// TwinCAT 3 PLC project EngineeringToolbox
// Title: EngineeringToolbox
// Company: Beckhoff Electronics Mfg
// Author: Daniel Schlingmann
// ProjectVersion: 3.1.2.4
// Description: Engineering Toolbox Library The library is provided "as-is" for TwinCAT3.1 by the Beckhoff Industry Management for Electronics Manufacturing. Please check the function "DisclaimerStatement : WSTRING[1500]" in additon to the following disclaimer: THE SOFTWARE IS PROVIDED "AS IS", WITHOUT WARRANTY OF ANY KIND, EXPRESS OR IMPLIED, INCLUDING BUT NOT LIMITED TO THE WARRANTIES OF MERCHANTABILITY, FITNESS FOR A PARTICULAR PURPOSE AND NONINFRINGEMENT. IN NO EVENT SHALL THE AUTHORS OR COPYRIGHT HOLDERS BE LIABLE FOR ANY CLAIM, DAMAGES OR OTHER LIABILITY, WHETHER IN AN ACTION OF CONTRACT, TORT OR OTHERWISE, ARISING FROM, OUT OF OR IN CONNECTION WITH THE SOFTWARE OR THE USE OR OTHER DEALINGS IN THE SOFTWARE.
// ProgramVersion: 3.1.4022.7
// libraries:
//   Tc2_Drive, * (Beckhoff Automation GmbH)
//   Tc2_EtherCAT, * (Beckhoff Automation GmbH)
//   Tc2_IoFunctions, * (Beckhoff Automation GmbH)
//   Tc2_Math, * (Beckhoff Automation GmbH)
//   Tc2_MC2, * (Beckhoff Automation GmbH)
//   Tc2_MC2_Camming, * (Beckhoff Automation GmbH)
//   Tc2_MC2_Drive, * (Beckhoff Automation GmbH)
//   Tc2_MC2_FlyingSaw, * (Beckhoff Automation GmbH)
//   Tc2_MDP, * (Beckhoff Automation GmbH)
//   Tc2_ModbusRTU, * (Beckhoff Automation GmbH)
//   Tc2_ModbusSrv, * (Beckhoff Automation GmbH)
//   Tc2_NC, * (Beckhoff Automation GmbH)
//   Tc2_NCI, * (Beckhoff Automation GmbH)
//   Tc2_NcKinematicTransformation, * (Beckhoff Automation GmbH)
//   Tc2_PlcInterpolation, * (Beckhoff Automation GmbH)
//   Tc2_SerialCom, * (Beckhoff Automation GmbH)
//   Tc2_Smtp, * (Beckhoff Automation GmbH)
//   Tc2_Standard, * (Beckhoff Automation GmbH)
//   Tc2_SUPS, * (Beckhoff Automation GmbH)
//   Tc2_System, * (Beckhoff Automation GmbH)
//   Tc2_TcpIp, * (Beckhoff Automation GmbH)
//   Tc2_Utilities, * (Beckhoff Automation GmbH)
//   Tc2_XmlDataSrv, * (Beckhoff Automation GmbH)
//   Tc3_Module, * (Beckhoff Automation GmbH)
//   Tc2_BackupRestoreEL6900,newest,Beckhoff Automation GmbH
// project tree:
//   GVLs/ Gvl.TcGVL (not stored), PARAM.TcGVL (not stored)
//   POUs/BoundsCheck/ boundsError.TcPOU (not stored), boundsOK.TcPOU (not stored), checkBounds.TcPOU (not stored), CheckBoundsInfo.TcPOU (not stored)
//   POUs/Connectivity/ADS/ AdsDataExchange.TcPOU (not stored)
//   POUs/Connectivity/ Ipv4Addr_TO_UDINT.TcPOU (not stored), U_DEVICE_COM_CACHE.TcDUT (not stored), U_IPv4Addr.TcDUT, isValidIPv4Addr.TcPOU (not stored)
//   POUs/Connectivity/TF6310-TcpServer/DeviceCom/ TCPDeviceCom_SendRecBytes.TcPOU (not stored), TCPDeviceCom_SendRecString.TcPOU (not stored)
//   POUs/Connectivity/TF6340-SerialCom/ComPortDeviceCom/ ComPortDeviceCom_BufferHandle.TcPOU (not stored), ComPortDeviceCom_SendRecBytes.TcPOU (not stored), ComPortDeviceCom_SendRecString.TcPOU, ComPortEL6x22BEasyConnect.TcPOU
//   POUs/Connectivity/TF6340-SerialCom/ComPortBasic/ ComPortBackground.TcPOU, ComPortSendRec.TcPOU (not stored)
//   POUs/Connectivity/TF625x-Modbus/Master/TF6250-ModbusTcpServer/TCP/ ModbusTcpMaster.TcPOU
//   POUs/Connectivity/TF625x-Modbus/Master/TF6250-ModbusTcpServer/UDP/ ModbusUdpMaster.TcPOU (not stored)
//   POUs/Connectivity/TF625x-Modbus/Master/TF6255-ModbusRtu/ ModbusRtuMaster22B.TcPOU, ModbusRtuMaster5B.TcPOU, ModbusRtuMasterPC.TcPOU (not stored)
//   POUs/Connectivity/TF625x-Modbus/Master/_Components/ ModbusJob.TcPOU (not stored), ModbusSlaveCom.TcPOU (not stored)
//   POUs/Connectivity/TF625x-Modbus/Slave/ ModbusSlaveBase.TcPOU (not stored)
//   POUs/Connectivity/TF6310-TcpServer/TcpBasic/ TCPSendRecCtrl.TcPOU, TCPConnectionCtrl.TcPOU (not stored), TCPSocketCtrl.TcPOU (not stored)
//   POUs/Connectivity/TF6310-TcpServer/UdpBasic/ UDPSendRecCtrl.TcPOU (not stored), UDPServerCtrl.TcPOU, UDPSocketCtrl.TcPOU (not stored)
//   POUs/ControllerTools/ AverageFilter.TcPOU (not stored), PIDController.TcPOU, PT1Filter.TcPOU (not stored), signum.TcPOU, SlewRateLimitter.TcPOU (not stored), SlidingAverageExt.TcPOU (not stored), SlidingAverage.TcPOU (not stored), ThreePointController.TcPOU (not stored)
//   POUs/DataBuffer/ DoubleBuffer.TcPOU, Quicksort.TcPOU
//   POUs/DataBuffer/FiFo/ Fifo.TcPOU, FiFoExt.TcPOU, FiFoLRealSimple.TcPOU, FiFoBase.TcPOU (not stored)
//   POUs/DataBuffer/LiFo/ LiFoBase.TcPOU (not stored), LiFoExt.TcPOU, LiFo.TcPOU (not stored)
//   POUs/DataBuffer/Ringbuffer/ RingbufferBase.TcPOU (not stored), Ringbuffer.TcPOU, RingbufferCharSimple.TcPOU, RingbufferExt.TcPOU (not stored), RingbufferByteSimple.TcPOU, RingbufferLRealSimple.TcPOU (not stored), RingbufferRealSimple.TcPOU (not stored)
//   POUs/EventLogger/ EventsWriteToLogbook.TcPOU (not stored), EVENT_HANDLING_CONFIG.TcDUT, getEventClassPriority.TcPOU (not stored), getEventClassText.TcPOU (not stored), SOURCE_ID.TcDUT
//   POUs/EventLogger/ReadEvents/ EventlogRead.TcPOU (not stored), EVENTLOG_READ_DATA.TcDUT, EVENTLOG_READ_HANDLEINFO.TcDUT, EVENTLOG_READ_STREAM.TcDUT (not stored), EVENTLOG_READ_STREAM_DATA_RAW.TcDUT (not stored), EVENTLOG_READ_STREAM_DATA_RAW_EX.TcDUT (not stored)
//   POUs/EventLogger/TriggerEvents/ EventHandling.TcPOU (not stored), EventHandlingGrp10.TcPOU (not stored), EventHandlingGrp25.TcPOU (not stored), EventHandlingGrp50.TcPOU, EventHandlingGrpCustomized.TcPOU (not stored), EventHandlingConfirmIsReq.TcPOU (not stored), EventHandlingStatisticInfo.TcPOU (not stored)
//   POUs/Fieldbus/CANopen/ CANopenMasterDiag.TcPOU, CANopenMasterIO.TcPOU (not stored)
//   POUs/Fieldbus/EAP/ EAP_PUB_SUB_IO.TcPOU (not stored), EAP_DEVICE_IO.TcPOU, EAP_PUB_VAR.TcPOU (not stored), EAP_SUB_VAR.TcPOU
//   POUs/Fieldbus/EtherCAT/ EcCoEReadNewestDiagMsg.TcPOU (not stored), EcDiagBase.TcPOU (not stored), EcDiagBase_wEvents.TcPOU (not stored)
//   POUs/Fieldbus/EtherCAT/_Components/ EcMasterIO.TcPOU, EcMasterSupervisor.TcPOU (not stored), EcSlavesDiag.TcPOU (not stored), EcSlaveSupervisor.TcPOU (not stored), EC_MASTER_DEVICE_STATE.TcDUT (not stored), EC_SLAVE_DIAG_INFO_DATA.TcDUT (not stored)
//   POUs/Fieldbus/Profibus/ ProfibusMasterDiag.TcPOU (not stored), ProfibusMasterIO.TcPOU (not stored)
//   POUs/Fieldbus/Profinet/ ProfinetControllerIO.TcPOU (not stored), ProfinetControllerIO_wEvents.TcPOU (not stored), ProfinetDeviceIO.TcPOU (not stored)
//   POUs/FileHandling/Basic/ FileHandling.TcPOU (not stored), ReadDirSimple.TcPOU (not stored), ReadDirSimpleExt.TcPOU (not stored)
//   POUs/FileHandling/TF6421-XmlServer/ XmlReadWrite.TcPOU (not stored), XmlReadWriteWithBackupFile.TcPOU
//   POUs/IO/Analog/ AnalogIn.TcPOU (not stored), AnalogIn32.TcPOU (not stored), AnalogInELMBase.TcPOU, AnalogInELMSingleSampleDINT.TcPOU (not stored), AnalogInELMSingleSampleREAL.TcPOU (not stored), AnalogInREAL.TcPOU (not stored), AnalogOut.TcPOU (not stored)
//   POUs/IO/ BlowOffSensors.TcPOU (not stored), Button.TcPOU (not stored), ButtonExt.TcPOU (not stored), Fuse.TcPOU, InOut.TcPOU, InOutExt.TcPOU (not stored), Input.TcPOU, Output.TcPOU (not stored)
//   POUs/IO/Cylinder/ Cylinder.TcPOU, CylinderExt.TcPOU (not stored), CylinderType4.TcPOU, I_Cylinder.TcIO
//   POUs/IO/Drives/ AxDriveBase.TcPOU (not stored), AxDriveGetRef.TcPOU (not stored), I_AxDriveBase.TcIO (not stored)
//   POUs/IO/Drives/CoE/ AxDriveCoE.TcPOU, AxDriveCoE_wEvents.TcPOU (not stored), CiA_DS402Controlword.TcPOU (not stored), CiA_DS402Statusword.TcPOU, eCiA_DS402_CONTROL_CMD.TcDUT (not stored), eCiA_DS402_STATUS_STATE.TcDUT (not stored)
//   POUs/IO/Drives/CoE/EL72xx/ AxDriveCoE_EL72xxParam.TcPOU, CiA_DS402StatuswordEx7xxx.TcPOU (not stored)
//   POUs/IO/Drives/DC/Ey73xx/ AxDriveDC.TcPOU (not stored), AxDriveDC_wEvents.TcPOU (not stored)
//   POUs/IO/Drives/SoE/ AxDriveSoE_Ax5000CommutationCalib.TcPOU, AxDriveSoE_Ax5000CalcPower.TcPOU (not stored), AxDriveSoE_Ax5000SwitchParamSet.TcPOU, Ax580x.TcPOU (not stored), AxDriveSoE_Ax5000.TcPOU (not stored), AxDriveSoE_Ax5000Param.TcPOU (not stored), AxDriveSoE_Ax5000wEvents.TcPOU (not stored), AxDriveSoE_Rexroth.TcPOU (not stored)
//   POUs/IO/Drives/SoE/Ax5000ParamSTRUCTs/P/ AX5000_P_0001.TcDUT, AX5000_P_0002.TcDUT, AX5000_P_0003.TcDUT, AX5000_P_0004.TcDUT, AX5000_P_0009.TcDUT (not stored), AX5000_P_0010.TcDUT (not stored), AX5000_P_0020.TcDUT (not stored), AX5000_P_0021.TcDUT (not stored), AX5000_P_0040.TcDUT (not stored), AX5000_P_0050.TcDUT (not stored), AX5000_P_0051.TcDUT (not stored), AX5000_P_0052.TcDUT (not stored), AX5000_P_0053.TcDUT (not stored), AX5000_P_0054.TcDUT, AX5000_P_0055.TcDUT, AX5000_P_0056.TcDUT (not stored), AX5000_P_0057.TcDUT (not stored), AX5000_P_0058.TcDUT (not stored), AX5000_P_0059.TcDUT (not stored), AX5000_P_0060.TcDUT, AX5000_P_0061.TcDUT (not stored), AX5000_P_0062.TcDUT, AX5000_P_0063.TcDUT (not stored), AX5000_P_0064.TcDUT, AX5000_P_0065.TcDUT (not stored), AX5000_P_0066.TcDUT (not stored), AX5000_P_0067.TcDUT (not stored), AX5000_P_0068.TcDUT, AX5000_P_0069.TcDUT (not stored), AX5000_P_0070.TcDUT (not stored), AX5000_P_0071.TcDUT (not stored), AX5000_P_0072.TcDUT (not stored), AX5000_P_0073.TcDUT (not stored), AX5000_P_0074.TcDUT, AX5000_P_0075.TcDUT, AX5000_P_0076.TcDUT, AX5000_P_0077.TcDUT, AX5000_P_0078.TcDUT (not stored), AX5000_P_0088.TcDUT (not stored), AX5000_P_0089.TcDUT, AX5000_P_0090.TcDUT, AX5000_P_0091.TcDUT, AX5000_P_0092.TcDUT (not stored), AX5000_P_0093.TcDUT (not stored), AX5000_P_0096.TcDUT, AX5000_P_0097.TcDUT (not stored), AX5000_P_0098_beckhoff.TcDUT, AX5000_P_0098_beckhoff_electrical_data.TcDUT, AX5000_P_0099.TcDUT, AX5000_P_0100.TcDUT, AX5000_P_0101.TcDUT (not stored), AX5000_P_0102.TcDUT (not stored), AX5000_P_0103.TcDUT, AX5000_P_0104.TcDUT (not stored), AX5000_P_0105.TcDUT, AX5000_P_0106.TcDUT (not stored), AX5000_P_0107.TcDUT, AX5000_P_0108.TcDUT (not stored), AX5000_P_0109.TcDUT, AX5000_P_0110.TcDUT (not stored), AX5000_P_0111.TcDUT, AX5000_P_0112.TcDUT, AX5000_P_0113.TcDUT (not stored), AX5000_P_0114.TcDUT (not stored), AX5000_P_0115.TcDUT, AX5000_P_0116.TcDUT (not stored), AX5000_P_0117.TcDUT, AX5000_P_0118.TcDUT (not stored), AX5000_P_0119.TcDUT (not stored), AX5000_P_0125.TcDUT (not stored), AX5000_P_0126.TcDUT (not stored), AX5000_P_0127.TcDUT (not stored), AX5000_P_0128.TcDUT (not stored), AX5000_P_0150.TcDUT (not stored), AX5000_P_0151.TcDUT, AX5000_P_0152.TcDUT (not stored), AX5000_P_0153.TcDUT, AX5000_P_0154.TcDUT (not stored), AX5000_P_0155.TcDUT, AX5000_P_0158.TcDUT (not stored), AX5000_P_0159.TcDUT (not stored), AX5000_P_0160.TcDUT (not stored), AX5000_P_0161.TcDUT (not stored), AX5000_P_0162.TcDUT (not stored), AX5000_P_0163.TcDUT (not stored), AX5000_P_0165.TcDUT, AX5000_P_0166.TcDUT (not stored), AX5000_P_0167.TcDUT, AX5000_P_0168.TcDUT, AX5000_P_0169.TcDUT (not stored), AX5000_P_0170.TcDUT (not stored), AX5000_P_0171.TcDUT, AX5000_P_0180.TcDUT (not stored), AX5000_P_0181.TcDUT (not stored), AX5000_P_0182.TcDUT, AX5000_P_0183.TcDUT (not stored), AX5000_P_0184.TcDUT (not stored), AX5000_P_0185.TcDUT, AX5000_P_0188.TcDUT (not stored), AX5000_P_0189.TcDUT (not stored), AX5000_P_0192.TcDUT, AX5000_P_0193.TcDUT, AX5000_P_0196.TcDUT (not stored), AX5000_P_0198.TcDUT (not stored), AX5000_P_0199.TcDUT, AX5000_P_0200.TcDUT (not stored), AX5000_P_0201.TcDUT (not stored), AX5000_P_0202.TcDUT (not stored), AX5000_P_0203.TcDUT (not stored), AX5000_P_0204.TcDUT (not stored), AX5000_P_0205.TcDUT (not stored), AX5000_P_0206.TcDUT (not stored), AX5000_P_0207.TcDUT (not stored), AX5000_P_0208.TcDUT (not stored), AX5000_P_0209.TcDUT (not stored), AX5000_P_0210.TcDUT (not stored), AX5000_P_0211.TcDUT (not stored), AX5000_P_0212.TcDUT (not stored), AX5000_P_0213.TcDUT (not stored), AX5000_P_0214.TcDUT (not stored), AX5000_P_0215.TcDUT (not stored), AX5000_P_0216.TcDUT, AX5000_P_0217.TcDUT (not stored), AX5000_P_0218.TcDUT, AX5000_P_0219.TcDUT (not stored), AX5000_P_0220.TcDUT (not stored), AX5000_P_0221.TcDUT, AX5000_P_0250.TcDUT, AX5000_P_0251.TcDUT (not stored), AX5000_P_0252.TcDUT (not stored), AX5000_P_0253.TcDUT (not stored), AX5000_P_0254.TcDUT (not stored), AX5000_P_0255.TcDUT (not stored), AX5000_P_0256.TcDUT (not stored), AX5000_P_0270.TcDUT (not stored), AX5000_P_0271.TcDUT, AX5000_P_0272.TcDUT, AX5000_P_0273.TcDUT (not stored), AX5000_P_0274.TcDUT (not stored), AX5000_P_0275.TcDUT (not stored), AX5000_P_0276.TcDUT (not stored), AX5000_P_0277.TcDUT, AX5000_P_0278.TcDUT, AX5000_P_0300.TcDUT, AX5000_P_0301.TcDUT (not stored), AX5000_P_0302.TcDUT (not stored), AX5000_P_0303.TcDUT (not stored), AX5000_P_0304.TcDUT (not stored), AX5000_P_0305.TcDUT (not stored), AX5000_P_0306.TcDUT, AX5000_P_0307.TcDUT, AX5000_P_0308.TcDUT (not stored), AX5000_P_0309.TcDUT, AX5000_P_0310.TcDUT (not stored), AX5000_P_0311.TcDUT (not stored), AX5000_P_0312.TcDUT (not stored), AX5000_P_0313.TcDUT (not stored), AX5000_P_0314.TcDUT (not stored), AX5000_P_0315.TcDUT (not stored), AX5000_P_0316.TcDUT (not stored), AX5000_P_0317.TcDUT, AX5000_P_0320.TcDUT (not stored), AX5000_P_0321.TcDUT, AX5000_P_0322.TcDUT, AX5000_P_0323.TcDUT (not stored), AX5000_P_0324.TcDUT (not stored), AX5000_P_0325.TcDUT (not stored), AX5000_P_0326.TcDUT, AX5000_P_0350.TcDUT (not stored), AX5000_P_0351.TcDUT (not stored), AX5000_P_0352.TcDUT (not stored), AX5000_P_0353.TcDUT, AX5000_P_0354.TcDUT (not stored), AX5000_P_0356.TcDUT (not stored), AX5000_P_0360.TcDUT (not stored), AX5000_P_0361.TcDUT, AX5000_P_0400.TcDUT, AX5000_P_0401.TcDUT, AX5000_P_0402.TcDUT (not stored), AX5000_P_0451.TcDUT (not stored), AX5000_P_0452.TcDUT, AX5000_P_0453.TcDUT, AX5000_P_0454.TcDUT (not stored), AX5000_P_0455.TcDUT, AX5000_P_0456.TcDUT (not stored), AX5000_P_0457.TcDUT (not stored), AX5000_P_0458.TcDUT (not stored), AX5000_P_0459.TcDUT (not stored), AX5000_P_0460.TcDUT, AX5000_P_0461.TcDUT (not stored), AX5000_P_0462.TcDUT, AX5000_P_0463.TcDUT, AX5000_P_0464.TcDUT (not stored), AX5000_P_0502.TcDUT, AX5000_P_0503.TcDUT (not stored), AX5000_P_0504.TcDUT (not stored), AX5000_P_0505.TcDUT (not stored), AX5000_P_0511.TcDUT (not stored), AX5000_P_0512.TcDUT (not stored), AX5000_P_0513.TcDUT, AX5000_P_0514.TcDUT (not stored), AX5000_P_0515.TcDUT (not stored), AX5000_P_0516.TcDUT (not stored), AX5000_P_0517.TcDUT (not stored), AX5000_P_0518.TcDUT (not stored), AX5000_P_0552.TcDUT, AX5000_P_0553.TcDUT (not stored), AX5000_P_0554.TcDUT (not stored), AX5000_P_0555.TcDUT, AX5000_P_0556.TcDUT (not stored), AX5000_P_0557.TcDUT (not stored), AX5000_P_0558.TcDUT, AX5000_P_0601.TcDUT (not stored), AX5000_P_0602.TcDUT (not stored), AX5000_P_0610.TcDUT (not stored), AX5000_P_0611.TcDUT, AX5000_P_0800.TcDUT (not stored), AX5000_P_0801.TcDUT (not stored), AX5000_P_0802.TcDUT, AX5000_P_0804.TcDUT (not stored), AX5000_P_0805.TcDUT (not stored), AX5000_P_0806.TcDUT (not stored), AX5000_P_0810.TcDUT, AX5000_P_0811.TcDUT (not stored), AX5000_P_0850.TcDUT (not stored), AX5000_P_0851.TcDUT (not stored), AX5000_P_0900.TcDUT (not stored), AX5000_P_0901.TcDUT, AX5000_P_0902.TcDUT (not stored), AX5000_P_0904.TcDUT, AX5000_P_0905.TcDUT (not stored), AX5000_P_0906.TcDUT, AX5000_P_0912.TcDUT (not stored), AX5000_P_1000.TcDUT (not stored), AX5000_P_1001.TcDUT (not stored), AX5000_P_1002.TcDUT, AX5000_P_1003.TcDUT, AX5000_P_1004.TcDUT (not stored), AX5000_P_1005.TcDUT, AX5000_P_1006.TcDUT, AX5000_P_1007.TcDUT (not stored), AX5000_P_1008.TcDUT (not stored), AX5000_P_1009.TcDUT (not stored), AX5000_P_1010.TcDUT (not stored), AX5000_P_1011.TcDUT, AX5000_P_1012.TcDUT, AX5000_P_1020.TcDUT, AX5000_P_1021.TcDUT, AX5000_P_1022.TcDUT (not stored), AX5000_P_2000.TcDUT (not stored), AX5000_P_2001.TcDUT (not stored), AX5000_P_2002.TcDUT (not stored)
//   POUs/IO/Drives/SoE/Ax5000ParamSTRUCTs/S/ AX5000_S_0001.TcDUT (not stored), AX5000_S_0002.TcDUT, AX5000_S_0007.TcDUT (not stored), AX5000_S_0011.TcDUT (not stored), AX5000_S_0012.TcDUT, AX5000_S_0013.TcDUT (not stored), AX5000_S_0015.TcDUT (not stored), AX5000_S_0016.TcDUT (not stored), AX5000_S_0017.TcDUT, AX5000_S_0018.TcDUT (not stored), AX5000_S_0024.TcDUT (not stored), AX5000_S_0029.TcDUT (not stored), AX5000_S_0030.TcDUT (not stored), AX5000_S_0031.TcDUT (not stored), AX5000_S_0032.TcDUT (not stored), AX5000_S_0033.TcDUT, AX5000_S_0034.TcDUT, AX5000_S_0035.TcDUT (not stored), AX5000_S_0036.TcDUT (not stored), AX5000_S_0037.TcDUT (not stored), AX5000_S_0040.TcDUT, AX5000_S_0043.TcDUT, AX5000_S_0044.TcDUT, AX5000_S_0045.TcDUT, AX5000_S_0046.TcDUT, AX5000_S_0047.TcDUT, AX5000_S_0048.TcDUT (not stored), AX5000_S_0051.TcDUT (not stored), AX5000_S_0053.TcDUT (not stored), AX5000_S_0055.TcDUT (not stored), AX5000_S_0076.TcDUT (not stored), AX5000_S_0079.TcDUT, AX5000_S_0080.TcDUT (not stored), AX5000_S_0081.TcDUT (not stored), AX5000_S_0082.TcDUT (not stored), AX5000_S_0083.TcDUT (not stored), AX5000_S_0084.TcDUT, AX5000_S_0085.TcDUT, AX5000_S_0086.TcDUT (not stored), AX5000_S_0091.TcDUT (not stored), AX5000_S_0092.TcDUT (not stored), AX5000_S_0095.TcDUT (not stored), AX5000_S_0099.TcDUT (not stored), AX5000_S_0100.TcDUT (not stored), AX5000_S_0101.TcDUT (not stored), AX5000_S_0103.TcDUT, AX5000_S_0104.TcDUT (not stored), AX5000_S_0106.TcDUT (not stored), AX5000_S_0107.TcDUT, AX5000_S_0109.TcDUT (not stored), AX5000_S_0110.TcDUT (not stored), AX5000_S_0111.TcDUT (not stored), AX5000_S_0112.TcDUT (not stored), AX5000_S_0113.TcDUT, AX5000_S_0119.TcDUT (not stored), AX5000_S_0120.TcDUT (not stored), AX5000_S_0124.TcDUT (not stored), AX5000_S_0126.TcDUT (not stored), AX5000_S_0130.TcDUT, AX5000_S_0131.TcDUT (not stored), AX5000_S_0134.TcDUT (not stored), AX5000_S_0135.TcDUT (not stored), AX5000_S_0136.TcDUT (not stored), AX5000_S_0137.TcDUT (not stored), AX5000_S_0143.TcDUT (not stored), AX5000_S_0149.TcDUT (not stored), AX5000_S_0159.TcDUT (not stored), AX5000_S_0160.TcDUT (not stored), AX5000_S_0161.TcDUT (not stored), AX5000_S_0162.TcDUT (not stored), AX5000_S_0163.TcDUT (not stored), AX5000_S_0169.TcDUT, AX5000_S_0170.TcDUT, AX5000_S_0179.TcDUT (not stored), AX5000_S_0185.TcDUT (not stored), AX5000_S_0186.TcDUT, AX5000_S_0187.TcDUT (not stored), AX5000_S_0188.TcDUT (not stored), AX5000_S_0189.TcDUT (not stored), AX5000_S_0196.TcDUT, AX5000_S_0200.TcDUT (not stored), AX5000_S_0201.TcDUT (not stored), AX5000_S_0203.TcDUT, AX5000_S_0204.TcDUT, AX5000_S_0206.TcDUT, AX5000_S_0207.TcDUT, AX5000_S_0216.TcDUT (not stored), AX5000_S_0217.TcDUT (not stored), AX5000_S_0219.TcDUT (not stored), AX5000_S_0254.TcDUT (not stored), AX5000_S_0256.TcDUT (not stored), AX5000_S_0257.TcDUT (not stored), AX5000_S_0267.TcDUT (not stored), AX5000_S_0273.TcDUT, AX5000_S_0274.TcDUT (not stored), AX5000_S_0292.TcDUT (not stored), AX5000_S_0295.TcDUT (not stored), AX5000_S_0296.TcDUT (not stored), AX5000_S_0347.TcDUT (not stored), AX5000_S_0348.TcDUT (not stored), AX5000_S_0372.TcDUT (not stored), AX5000_S_0374.TcDUT (not stored), AX5000_S_0375.TcDUT (not stored), AX5000_S_0380.TcDUT (not stored), AX5000_S_0381.TcDUT, AX5000_S_0383.TcDUT (not stored), AX5000_S_0384.TcDUT (not stored), AX5000_S_0390.TcDUT (not stored), AX5000_S_0403.TcDUT, AX5000_S_0405.TcDUT, AX5000_S_0409.TcDUT (not stored), AX5000_S_0410.TcDUT (not stored), AX5000_S_0429.TcDUT (not stored), AX5000_S_0432.TcDUT, AX5000_S_0435.TcDUT (not stored), AX5000_S_0436.TcDUT
//   POUs/IO/Drives/Stepper/ AxDriveStepper.TcPOU (not stored), AxDriveStepperParam.TcPOU (not stored), AxDriveStepper_wEvents.TcPOU (not stored)
//   POUs/IO/EL-EP/ AnalogOut_EL2535.TcPOU (not stored), EL1262_Base.TcPOU, EL3681.TcPOU (not stored), EL1904.TcPOU (not stored), EL69xx.TcPOU (not stored), EL3356.TcPOU, Eyx9xx.TcPOU (not stored), ZB8610.TcPOU (not stored)
//   POUs/IO/EL-EP/EL9x/ EL9501.TcPOU, EL9576.TcPOU (not stored), EL95xxPowerTerminal.TcPOU (not stored), ELSystemTerminal.TcPOU (not stored)
//   POUs/IO/_EcSlaveFWUpdater/ EcSlaveDevFWUpdater.TcPOU (not stored)
//   POUs/IO/_EcSlaveInfoDataIO/ EcSlaveInfoData.TcPOU (not stored), EcSlaveInfoDataExt.TcPOU, I_EcSlaveInfoData.TcIO (not stored)
//   POUs/IO/EL-EP/EL3403/ EL3403.TcPOU (not stored), EL3403Logic.TcPOU (not stored)
//   POUs/IO/EL-EP/EP92xxPwrBox/ EP9214.TcPOU (not stored), EP9214_CHANNEL.TcPOU, EP9224_0037.TcPOU (not stored), EP9224_0037_CHANNEL.TcPOU (not stored)
//   POUs/IO/FreqConv/EtherCAT/DS402/ EcFcDS402_ComBase.TcPOU (not stored)
//   POUs/IO/FreqConv/ IOFcCom.TcPOU (not stored)
//   POUs/IO/Motors/ IOMotor.TcPOU, IOMotor2Dir.TcPOU (not stored), IOMotorStarDelta.TcPOU (not stored)
//   POUs/IO/[underDev]/ Cylinder_wUnitItf.TcPOU (not stored)
//   POUs/IO/_ItfActuators/ I_ActuatorBase.TcIO, I_ActuatorEnableDisable.TcIO, I_ActuatorFwdRev.TcIO (not stored), I_ActuatorFwdBwd.TcIO (not stored), I_ActuatorLeftRight.TcIO (not stored), I_ActuatorOnOff.TcIO (not stored), I_ActuatorOpenClose.TcIO, I_ActuatorPosNeg.TcIO (not stored), I_ActuatorStartStop.TcIO (not stored), I_ActuatorUpDown.TcIO (not stored), I_ActuatorWorkBase.TcIO
//   POUs/IpcDiag/MDP/InfoModuls/ MDP_CPU.TcPOU (not stored), MDP_Fan.TcPOU (not stored), MDP_Mainboard.TcPOU, MDP_RaidSimple.TcPOU (not stored), MDP_ReadModulList.TcPOU, MDP_SiliconDrives.TcPOU (not stored), MDP_UPS.TcPOU
//   POUs/IpcDiag/MDP/ MDP_Info.TcPOU (not stored), MDP_IpcDiag.TcPOU, MDP_IpcDiag_wEvents.TcPOU (not stored)
//   POUs/IpcDiag/ UPSStatus.TcPOU
//   POUs/Logging/ DataFileLogger.TcPOU (not stored), DataUdpLogger.TcPOU, I_LogbookSubscriber.TcIO (not stored), I_Logbook.TcIO (not stored), Logbook.TcPOU (not stored), LogbookData.TcDUT (not stored), LogbookPuplisher.TcPOU (not stored), LogbookSubEventLog.TcPOU (not stored), LogbookSubSendMail.TcPOU (not stored), adsLogError.TcPOU (not stored), adsLogHint.TcPOU, adsLogWarn.TcPOU (not stored), LogbookSubSysLog.TcPOU (not stored), LogbookSubWriteFile.TcPOU (not stored), Logbook_wEventClass.TcPOU (not stored), adsLogwTcEventClass.TcPOU (not stored)
//   POUs/Motion/TF50xx-NC/00_Base/ I_AxNcPTP.TcIO, AxFbBase.TcPOU (not stored), AxRWParaBase.TcPOU (not stored), I_AxNcBase.TcIO (not stored)
//   POUs/Motion/TF50xx-NC/02_Options/Parameter/ AxPara.TcPOU, AxParaCtrl.TcPOU (not stored)
//   POUs/Motion/TF50xx-NC/03_Utilities/ AxAutoWriteSoftLimit.TcPOU (not stored), CoordinateTransformation2D.TcPOU (not stored), AxCalcPosBias.TcPOU (not stored), AxResonanceAvoidance.TcPOU (not stored) (excluded from build), AxSoftSyncDistance.TcPOU (not stored), AxStatemodel.TcPOU (not stored), AxAutoFct.TcPOU, AX_JOB.TcPOU (not stored), getOvrVelo.TcPOU
//   POUs/Motion/TF50xx-NC/ AxNcPTPwJobs.TcPOU (not stored), AxNcBaseExt.TcPOU (not stored), AxNcPtpGear.TcPOU (not stored), AxNcBase.TcPOU (not stored), AxNcPTP.TcPOU
//   POUs/Motion/TF5100-NCI/ NciChannel_wEvents.TcPOU, NciChannel.TcPOU
//   POUs/Motion/TF511x-KIN/03_DUTs/Positions/ KIN_POSITIONS.TcPOU, KIN_POSITIONS_ACS_DUT.TcDUT (not stored), KIN_POSITIONS_MCS_DUT.TcDUT (not stored), U_KIN_POSITIONS.TcDUT (not stored)
//   POUs/Motion/TF511x-KIN/03_DUTs/Trafo/ KIN_CALCTRAFO_AXPOS_PARAM.TcPOU, KIN_STATE_OBSERVER_OID_PARAM.TcPOU, KIN_STATICTRAFO_PARAM.TcPOU (not stored), KIN_TOOLTRAFO_PARAM.TcPOU (not stored), UCS.TcPOU (not stored)
//   POUs/Motion/ VALUE_3D.TcPOU (not stored), VALUE_3D_DUT.TcDUT (not stored), VALUE_6D.TcPOU (not stored), VALUE_6D_DUT.TcDUT (not stored)
//   POUs/Safety/Diag/ SafetyLogicAndIOTerminalDiag.TcPOU (not stored), SafetyIODeviceDiagRead.TcPOU, SafetyIODeviceDiag_wEvents.TcPOU (not stored), SafetyIOsDiag.TcPOU (not stored), SafetyLogicTerminalDiag.TcPOU (not stored), SafetyPlcTerminalDiag.TcPOU (not stored)
//   POUs/StringHelper/ CHR_TO_STR.TcPOU (not stored), cutStrNumberToSeperator.TcPOU, cutStrToSeperator2.TcPOU (not stored), replaceUmlauts.TcPOU (not stored), stringCmp.TcPOU (not stored), STR_TO_ASC.TcPOU, cutStrToSeperator.TcPOU (not stored), cutWStrToSeperator.TcPOU (not stored), DWORD_TO_BINSTR_EXT.TcPOU, DWORD_TO_HEXSTR_EXT.TcPOU (not stored), getCntCharInStr.TcPOU (not stored), getCntCharInWStr.TcPOU (not stored), isWStringNumeric.TcPOU, HEXSTR_TO_DWORD.TcPOU (not stored), HEXSTR_TO_LWORD.TcPOU (not stored), INSERT_EXT.TcPOU (not stored), LWORD_TO_BINSTR_EXT.TcPOU (not stored), LWORD_TO_HEXSTR_EXT.TcPOU (not stored), readStrToSeperator.TcPOU (not stored), replaceInString.TcPOU, getFilledString.TcPOU (not stored), isStringNumeric.TcPOU (not stored), readWStrToSeperator.TcPOU (not stored), replaceInWString.TcPOU (not stored), U_MAX_STRING.TcDUT (not stored), U_MAX_WSTRING.TcDUT (not stored), WINSERT_EXT.TcPOU
//   POUs/System/ SystemInfo.TcPOU, SystemInfo64.TcPOU (excluded from build), SystemPulses.TcPOU, TaskInfo.TcPOU
//   POUs/TimeHelper/ PartsPerTime.TcPOU, createTOD.TcPOU, getDateAndTimeDelta.TcPOU, getTonCountdown.TcPOU (not stored), LivebitCheck.TcPOU, Ontime.TcPOU, OntimeExt.TcPOU (not stored), OntimeSimple.TcPOU, Pulse.TcPOU (not stored), SensorTimeoutCheck.TcPOU (not stored), systemtimeInCam.TcPOU (not stored), systemtimeCmp.TcPOU, systemtimeInWin.TcPOU (not stored), TimeSwitch.TcPOU (not stored), TONRecord.TcPOU (not stored), TONTOF.TcPOU, VeloLinearMeasurement.TcPOU (not stored)
//   POUs/_Miscellaneous/64BitFunctions/ CLEARBIT64.TcPOU, CSETBIT64.TcPOU (not stored), GETBIT64.TcPOU (not stored), SETBIT64.TcPOU (not stored)
//   POUs/_Miscellaneous/Conversions/ TO_FMREAL.TcPOU (not stored), ADSERROR_TO_HRESULT.TcPOU, DWORD_TO_REAL_EX.TcPOU (not stored), HRESULT_TO_ADSERROR.TcPOU (not stored), REAL_TO_FMLREAL.TcPOU (not stored), LWORD_TO_LREAL_EX.TcPOU (not stored), SWAP_BYTES_OF_WORDS.TcPOU (not stored), SWAP_WORDS_OF_DWORD.TcPOU, SWAP_WORDS_OF_LWORD.TcPOU, ADSERROR_TO_WIN32ERROR.TcPOU (not stored), ADSERROR_TO_WSERROR.TcPOU (not stored), C_TO_F.TcPOU (not stored), DEGREES_TO_RPM.TcPOU (not stored), F_TO_C.TcPOU (not stored), GF_TO_N.TcPOU, TO_FMLREAL.TcPOU (not stored), MMIN_TO_MMS.TcPOU (not stored), MMS_TO_MMIN.TcPOU (not stored), N_TO_GF.TcPOU, RPM_TO_DEGREES.TcPOU (not stored)
//   POUs/_Miscellaneous/ nextIdx.TcPOU, scale2.TcPOU, TC_VN_COLORS.TcDUT (excluded from build), FbBase.TcPOU (not stored), CAM.TcPOU (not stored), CAM3D.TcPOU, COLOR.TcDUT, ERROR_HDL.TcPOU, FbBaseExt.TcPOU (not stored), FbBaseOutputs.TcPOU (not stored), getNoOfBits.TcPOU (not stored), LCID.TcDUT, eLCID.TcDUT (not stored), LOGx.TcPOU (not stored), OEECalculation.TcPOU (not stored), polynomial.TcPOU, RF_TRIG.TcPOU (not stored), scale.TcPOU (not stored), SEQUENCE_HDL.TcPOU (not stored), setNoOfBits.TcPOU (not stored), TEST_FB.TcPOU (not stored), TOGGLE.TcPOU, U_32BIT_DATATYPE.TcDUT (not stored), U_64BIT_DATATYPE.TcDUT (not stored), WIN.TcPOU
//   POUs/Safety/ SafetyCircuit.TcPOU (not stored), SafetyGroupIO.TcPOU, SafetyPlcBackupRestore.TcPOU, SAFETY_CIRCUIT_STATUS.TcDUT
//   POUs/Statemodel/control/ I_StatemodelBase.TcIO (not stored), I_Statemodel.TcIO (not stored), Statemodel.TcPOU (not stored)
//   POUs/Statemodel/ eMODE.TcDUT (not stored), eSTATE.TcDUT (not stored)
//   POUs/Statemodel/UnitTemplate/ I_Statemodel_Unit.TcIO (not stored), Statemodel_Unit.TcPOU (not stored)
//   POUs/Motion/TF50xx-NC/01_Main/ AxAdmin.TcPOU (not stored), AxHoming.TcPOU (not stored), AxMotion.TcPOU (not stored)
//   POUs/Motion/TF50xx-NC/02_Options/Motion/ AxSuperposition.TcPOU, AxMoveSinus.TcPOU, AxHomingOnBlock.TcPOU
//   POUs/Motion/TF5100-NCI/01_Main/ NciAdmin.TcPOU, NciGrp.TcPOU, NciItp.TcPOU (not stored), NciMotion.TcPOU (not stored), NCI_REF.TcPOU (not stored)
//   POUs/Motion/TF5100-NCI/02_Options/Error/ NciChnEventHandling.TcPOU, NciEventHandling.TcPOU
//   POUs/Motion/TF5100-NCI/02_Options/MFunctions/ NciMFnc.TcPOU
//   POUs/Motion/TF5100-NCI/02_Options/PlcItp/ NciCreateItpTable.TcPOU, NciCreateItpTableEntryTemplate.TcPOU (not stored)
//   POUs/Motion/TF5100-NCI/02_Options/RParameter/ NCiReadWriteRParam.TcPOU
//   POUs/Motion/TF511x-KIN/01_Main/ KinAdmin.TcPOU (not stored), KIN_REF.TcPOU (not stored)
//   POUs/Motion/TF511x-KIN/02_Options/ KinLockUnlockTrafoParam.TcPOU (not stored), KinWriteToolTrafoParam.TcPOU (not stored), KinWriteUCSTrafoParam.TcPOU (not stored)
//   POUs/Motion/TF511x-KIN/ KinChannel.TcPOU
//   POUs/Motion/TF50xx-NC/02_Options/Coupling/ AxCamming.TcPOU, AxFlyingSaw.TcPOU (not stored), AxGear.TcPOU (not stored)
//   POUs/Motion/TF50xx-NC/02_Options/Error/ AxNcEventHandling.TcPOU (not stored), AxEventHandling.TcPOU (not stored)
//   POUs/Motion/TF50xx-NC/02_Options/Phasing/ AxPhasing.TcPOU
//   POUs/Motion/TF50xx-NC/02_Options/TouchProbe/ AxTouchProbe.TcPOU
//   POUs/StringHelper/ExtendedString/ ExtString.TcPOU (not stored), ExtWString.TcPOU, T_EXT_STRING.TcDUT (not stored), T_EXT_WSTRING.TcDUT (not stored)
//   POUs/TimeHelper/Conversions/ FILETIME_TO_DATE.TcPOU (not stored), LREAL_TO_TIME_SEC.TcPOU (not stored), FILETIME_TO_TOD.TcPOU (not stored), SYSTEMTIME_TO_TIME.TcPOU, SYSTEMTIME_TO_TIME_EX.TcPOU (not stored), SYSTEMTIME_TO_TOD.TcPOU (not stored), SYSTEMTIME_TO_DATE.TcPOU (not stored), TIME_TO_FMRLREAL.TcPOU (not stored), TIME_TO_SYSTEMTIME.TcPOU
//   Version/ disclaimerStatement.TcPOU (not stored), Global_Version.TcGVL
// real-time tasks:
//   TASK PlcTask: cycle T#10ms, priority 20, ADS port 350

// ---- POUs/Connectivity/U_IPv4Addr.TcDUT
//IP v4 address as an union to provide the address in a UDINT and array format 
TYPE U_IPv4Addr : 
UNION
	Stacked 				: UDINT; //IPv4 address combined in a UDINT
	Bytes 					: T_IPv4AddrArr; //IPv4 address as an array 0..3 of Byte
END_UNION
END_TYPE

// ---- POUs/EventLogger/EVENT_HANDLING_CONFIG.TcDUT
{attribute 'hide'}
//Library Param structure for EventLogger related function blocks  
TYPE EVENT_HANDLING_CONFIG :
STRUCT
	GRP_CUSTOMISED_MAX_EVENT								:	INT(1..1000) ;
	
	EVENTLOG_READ_MSG_LEN_MIN								:	INT(0..1) ;
	EVENTLOG_READ_MSG_LEN_MAX								:	INT(0..2096) ;	
                                                                     
	EVENTLOG_READ_MAX_EVENTS								:	INT(1..1000) ;
	                                                            
	ENABLE_DYNAMIC_EVENT_MSG_FORMAT							:	BOOL	; //Enable to adjust the placeholder (format) of the event messages according the use of Parameter EventHandling.Text1,Text2 and pText3
	
	CLASS_NONE_QUIT_REQUIRED								:	BOOL     ;
	CLASS_MAINTENANCE_QUIT_REQUIRED							:	BOOL     ;
	CLASS_MESSAGE_QUIT_REQUIRED								:	BOOL     ;
	CLASS_HINT_QUIT_REQUIRED								:	BOOL     ;
	CLASS_STATEINFO_QUIT_REQUIRED							:	BOOL     ;
	CLASS_INSTRUCTION_QUIT_REQUIRED							:	BOOL     ;
	CLASS_WARNING_QUIT_REQUIRED								:	BOOL     ;
	CLASS_ALARM_QUIT_REQUIRED								:	BOOL     ;
	CLASS_PARAMERROR_QUIT_REQUIRED							:	BOOL     ;
	                                                    	             
	CLASS_NONE_PRIORITY										:	UINT(0..3); //1=high ...3=low 
	CLASS_MAINTENANCE_PRIORITY								:	UINT(0..3); //1=high ...3=low 
	CLASS_MESSAGE_PRIORITY									:	UINT(0..3); //1=high ...3=low 
	CLASS_HINT_PRIORITY										:	UINT(0..3); //1=high ...3=low 
	CLASS_STATEINFO_PRIORITY								:	UINT(0..3); //1=high ...3=low 
	CLASS_INSTRUCTION_PRIORITY								:	UINT(0..3); //1=high ...3=low 
	CLASS_WARNING_PRIORITY									:	UINT(0..3); //1=high ...3=low 
	CLASS_ALARM_PRIORITY									:	UINT(0..3); //1=high ...3=low 
	CLASS_PARAMERROR_PRIORITY								:	UINT(0..3); //1=high ...3=low 
END_STRUCT
END_TYPE

// ---- POUs/EventLogger/ReadEvents/EVENTLOG_READ_DATA.TcDUT
TYPE EVENTLOG_READ_DATA :
STRUCT
	eClass			: E_TcEventClass;	//See Beckhoff documentation for more information
	Computer		: STRING(80);		//Computer name of event source
	Timestamp		: T_DCTIME64;		//Timestamp in 64bit DC time format 
	TimestampDT		: DT;				//Timestamp in DATE_AND_TIME format 
	SourceId		: DWORD;			//Event Source ID
	id				: DWORD;			//Event number	
	State			: DWORD;			//Event state 
	Flags			: DWORD;			(*  TCEVENTFLAG_REQ=0x0001,
											TCEVENTFLAG_REQMUSTCON=0x0002,
											TCEVENTFLAG_CON=0x0004,
											TCEVENTFLAG_RESET=0x0008,
											TCEVENTFLAG_PRIOCLASS=0x0010,
											TCEVENTFLAG_FMTSELF=0x0020,
											TCEVENTFLAG_LOG=0x0040,
											TCEVENTFLAG_MSGBOX=0x0080,
											TCEVENTFLAG_SRCID=0x0100,
											TCEVENTFLAG_SELFRESET=0x0200,
											TCEVENTFLAG_TCID=0x0400,
											TCEVENTFLAG_SIGNAL=0x0800,
											TCEVENTFLAG_ADS=0x8000 *)
	Source			: WSTRING(40);		//Source name	
	MsgText			: WSTRING(255);		//Event message text in Unicode
	MegLen			: DWORD;			//Length of event message
END_STRUCT
END_TYPE

// ---- POUs/EventLogger/ReadEvents/EVENTLOG_READ_HANDLEINFO.TcDUT
TYPE EVENTLOG_READ_HANDLEINFO :
STRUCT
	Enum			: DWORD;
	Count			: DWORD;
END_STRUCT
END_TYPE

// ---- POUs/EventLogger/SOURCE_ID.TcDUT
{attribute 'qualified_only'}
//Predefined EventLogger Source Ids which collaborate to the default TcEventLogger Excel sheet   
//Most source IDs are already used as initial values for function blocks in this lib
TYPE SOURCE_ID :
STRUCT	
	TC_IO_MESSAGES			:	UDINT := 300;		//Reserved - TC3 default for TcIoMessages.xml
	TC_NC_MESSAGES			:	UDINT := 500;		//Reserved - TC3 default for TcNcMessages.xml
	TC_MIN_CNC_ERRORS		:	UDINT := 550;		//Reserved - TC3 default for TcCncErrors.xml
	TC_MAX_CNC_ERRORS		:	UDINT := 599;		//Reserved - TC3 default for TcCncErrors.xml
	TC_MIN_CNC_USER_EVENTS	:	UDINT := 650;		//Reserved - TC3 TcCncUserEvents.xml
	TC_MAX_CNC_USER_EVENTS	:	UDINT := 699;		//Reserved - TC3 TcCncUserEvents.xml
	TC_NC_DEF				:	UDINT := 700;		//Reserved - TC3 default for NCDefs.xml
	TC_NC_DEF_2				:	UDINT := 701;		//Reserved - TC3 default for NCDefs.xml
	
//	TcIoMessages.xml		:	UDINT := 300;		space - TC3 default 
//	TcNcMessages.xml		:	UDINT := 500;		space - TC3 default
//	TcCncErrors.xml			:	UDINT := 550-599;	space - TC3 default
//	TcCncUserEvents.xml		:	UDINT := 650-699;	space - TC3 default
//	NCDefs.xml				:	UDINT := 700-701;	space - NC Default
	
// 	General 0000- 0100
	GENERAL_STARTUP			:	UDINT := 100000;
	IPC_DIAG				:	UDINT := 100001;
	
// Safety 	0300-0399
	MIN_SAFETY_PLC_TERM_DIAG:	UDINT := 100300;
	MAX_SAFETY_PLC_TERM_DIAG:	UDINT := 100309;

	MIN_SAFETY_IO_TERM_DIAG	:	UDINT := 100310;
	MAX_SAFETY_IO_TERM_DIAG	:	UDINT := 100399;

// NC		1000-1999
	MIN_NC_AXIS				:	UDINT := 101000;	// NC Axis Min 
	MAX_NC_AXIS				:	UDINT := 101199;	// NC Axis Max
	
	MIN_NCI_GROUP			:	UDINT := 101200;	// NCI Groups Min 
	MAX_NCI_GROUP			:	UDINT := 101209;	// NCI Groups Max 
	
	MIN_KIN_GROUP			:	UDINT := 101210;	// Kinematik Groups Min 
	MAX_KIN_GROUP			:	UDINT := 101219;	// Kinematik Groups Max 
	
	MIN_XTS_GROUP			:	UDINT := 101220;	// XTS Groups Min 
	MAX_XTS_GROUP			:	UDINT := 101229;	// XTS Groups Max 
	
	MIN_CA_GROUP			:	UDINT := 101230;	// CA - Collision Avoidance Min 
	MAX_CA_GROUP			:	UDINT := 101239;	// CA - Collision Avoidance Max 
	
	MIN_PP_GROUP			:	UDINT := 101240;	// PP - Pick and Place Min 
	MAX_PP_GROUP			:	UDINT := 101249;	// PP - Pick and Place Max 

// Drives	2000-2999
	MIN_DRIVE_SOE			:	UDINT := 102000;	// Sercos Drive Min 
	MAX_DRIVE_SOE			:	UDINT := 102199;	// Sercos Drive Max 
	
	MIN_DRIVE_COE			:	UDINT := 102200;	// CanOpen Drive Min 
	MAX_DRIVE_COE			:	UDINT := 102399;	// CanOpen Drive Max 

	MIN_DRIVE_HYDR			:	UDINT := 102400;	// Hydraulic Drive Min 
	MAX_DRIVE_HYDR			:	UDINT := 102599;	// Hydraulic Drive Max 
	
	MIN_DRIVE_STEPPER		:	UDINT := 102600;	// Stepper Drive Min 
	MAX_DRIVE_STEPPER		:	UDINT := 102799;	// Stepper Drive Max 
	
// Fieldbus	3000-3099
	MIN_HW_EC_DIAG			:	UDINT := 103000;	// EtherCAT Master Min 
	MAX_HW_EC_DIAG			:	UDINT := 103009;	// EtherCAT Master Max 

	MIN_HW_CAN_DIAG			:	UDINT := 103010;	// CanOpen Master Min 
	MAX_HW_CAN_DIAG			:	UDINT := 103019;	// CanOpen Master Max 

	MIN_HW_PB_DIAG			:	UDINT := 103020;	// ProfiBus Master Min 
	MAX_HW_PB_DIAG			:	UDINT := 103029;	// ProfiBus Master Max 

	MIN_HW_PN_DIAG			:	UDINT := 103030;	// ProfiNet Master Min 
	MAX_HW_PN_DIAG			:	UDINT := 103039;	// ProfiNet Master Max 

	MIN_HW_DN_DIAG			:	UDINT := 103040;	// DeviceNet Master Min 
	MAX_HW_DN_DIAG			:	UDINT := 103049;	// DeviceNet Master Max 

	MIN_HW_S3_DIAG			:	UDINT := 103050;	// Sercos 3 Master Min 
	MAX_HW_S3_DIAG			:	UDINT := 103059;	// Sercos 3 Master Max 

	MIN_HW_LB_DIAG			:	UDINT := 103060;	// LightBus Master Min 
	MAX_HW_LB_DIAG			:	UDINT := 103069;	// LightBus Master Max 

	MIN_HW_IB_DIAG			:	UDINT := 103070;	// InterBus Master Min 
	MAX_HW_IB_DIAG			:	UDINT := 103079;	// InterBus Master Max 

	MIN_HW_EIP_DIAG			:	UDINT := 103080;	// Ethernet/IP Master Min 
	MAX_HW_EIP_DIAG			:	UDINT := 103089;	// Ethernet/IP Master Max 
	
END_STRUCT
END_TYPE

// ---- POUs/IO/Drives/SoE/Ax5000ParamSTRUCTs/P/AX5000_P_0001.TcDUT
TYPE AX5000_P_0001 :
STRUCT
	Schwitching_frequencyof_the_IGBT_module:UINT;
END_STRUCT
END_TYPE

// ---- POUs/IO/Drives/SoE/Ax5000ParamSTRUCTs/P/AX5000_P_0002.TcDUT
TYPE AX5000_P_0002 :
STRUCT
	Current_ctrl_cycle_time:UINT:=100;
END_STRUCT
END_TYPE

// ---- POUs/IO/Drives/SoE/Ax5000ParamSTRUCTs/P/AX5000_P_0003.TcDUT
TYPE AX5000_P_0003 :
STRUCT
	Velocity_crtl_cycle_time:UINT;
END_STRUCT
END_TYPE

// ---- POUs/IO/Drives/SoE/Ax5000ParamSTRUCTs/P/AX5000_P_0004.TcDUT
TYPE AX5000_P_0004 :
STRUCT
	Position_ctrl_cycle_time:UINT;
END_STRUCT
END_TYPE

// ---- POUs/IO/Drives/SoE/Ax5000ParamSTRUCTs/P/AX5000_P_0054.TcDUT
TYPE AX5000_P_0054 :
STRUCT
	Actual_lenght:UINT;
	Max_lenght:UINT;
	Configures_drive_type:STRING(29);
END_STRUCT
END_TYPE

// ---- POUs/IO/Drives/SoE/Ax5000ParamSTRUCTs/P/AX5000_P_0055.TcDUT
TYPE AX5000_P_0055 :
STRUCT
	Motor_EMK:WORD;	(*Decimal Point: 1 *)
END_STRUCT
END_TYPE

// ---- POUs/IO/Drives/SoE/Ax5000ParamSTRUCTs/P/AX5000_P_0060.TcDUT
TYPE AX5000_P_0060 :
STRUCT
	Motor_type_and_usage:WORD;	(* "0"-->no brake;standard holding brake, "1"-->currentless locked,standard holding brake, "16"-->no brake; Holding emergency break, "17"-->currentless locked, olding emergency break*)
//	{attribute 'hide'}
	rsvd:ARRAY[0..7] OF UINT;
END_STRUCT
END_TYPE

// ---- POUs/IO/Drives/SoE/Ax5000ParamSTRUCTs/P/AX5000_P_0062.TcDUT
TYPE AX5000_P_0062 :
STRUCT
	Actual_lenght:UINT;
	Max_lenght:UINT;
	Time_constant:UINT;
	Warning_limit:UINT;
	Error_limit:UINT;
	Reaktion:UINT;
END_STRUCT
END_TYPE

// ---- POUs/IO/Drives/SoE/Ax5000ParamSTRUCTs/P/AX5000_P_0064.TcDUT
TYPE AX5000_P_0064 :
STRUCT
	Actual_motorbrake_current:UINT;
END_STRUCT
END_TYPE

// ---- POUs/IO/Drives/SoE/Ax5000ParamSTRUCTs/P/AX5000_P_0068.TcDUT
TYPE AX5000_P_0068 :
STRUCT
	Actual_lenght:UINT;
	Max_lenght:UINT;
	Overload_factor:UINT;
	CRC16:UINT;
END_STRUCT
END_TYPE

// ---- POUs/IO/Drives/SoE/Ax5000ParamSTRUCTs/P/AX5000_P_0074.TcDUT
TYPE AX5000_P_0074 :
STRUCT
	Actual_lenght:UINT;
	Max_lenght:UINT;
	Iq: ARRAY [0..9] OF UDINT;
	M: ARRAY [0..9] OF UDINT;
END_STRUCT
END_TYPE

// ---- POUs/IO/Drives/SoE/Ax5000ParamSTRUCTs/P/AX5000_P_0075.TcDUT
TYPE AX5000_P_0075 :
STRUCT
	Actual_lenght:UINT;
	Max_lenght:UINT;
	Iq: ARRAY[0..9] OF UDINT;
	Lq:ARRAY[0..9] OF UDINT;
END_STRUCT
END_TYPE

// ---- POUs/IO/Drives/SoE/Ax5000ParamSTRUCTs/P/AX5000_P_0076.TcDUT
TYPE AX5000_P_0076 :
STRUCT
	Actual_lenght:UINT;
	Max_lenght:UINT;
	Temperature:ARRAY [0..9] OF UINT;
	Resistance:ARRAY [0..9] OF UINT;
END_STRUCT
END_TYPE

// ---- POUs/IO/Drives/SoE/Ax5000ParamSTRUCTs/P/AX5000_P_0077.TcDUT
TYPE AX5000_P_0077 :
STRUCT
	Motor_rated_voltage:UINT;
END_STRUCT
END_TYPE

// ---- POUs/IO/Drives/SoE/Ax5000ParamSTRUCTs/P/AX5000_P_0089.TcDUT
TYPE AX5000_P_0089 :
STRUCT
	Actual_lenght:UINT;
	Max_lenght:UINT;
	IDN:UDINT;
	MinValue:UDINT;
	MaxValue:UDINT;
	IDN2:UDINT;
	MinValue2:UDINT;
	MaxValue2:UDINT;
	IDN3:UDINT;
	MinValue3:UDINT;
	MaxValue3:UDINT;
END_STRUCT
END_TYPE

// ---- POUs/IO/Drives/SoE/Ax5000ParamSTRUCTs/P/AX5000_P_0090.TcDUT
TYPE AX5000_P_0090 :
STRUCT
	Channel_peak_current:UDINT;
END_STRUCT
END_TYPE

// ---- POUs/IO/Drives/SoE/Ax5000ParamSTRUCTs/P/AX5000_P_0091.TcDUT
TYPE AX5000_P_0091 :
STRUCT
	Channel_rated_current:UDINT;
END_STRUCT
END_TYPE

// ---- POUs/IO/Drives/SoE/Ax5000ParamSTRUCTs/P/AX5000_P_0096.TcDUT
TYPE AX5000_P_0096 :
STRUCT
	Motor_brake_force_lock:BOOL;
	Motor_brake_force_unlock:BOOL;
//	{attribute 'hide'}
	Rsvd:ARRAY[0..13] OF BOOL;
END_STRUCT
END_TYPE

// ---- POUs/IO/Drives/SoE/Ax5000ParamSTRUCTs/P/AX5000_P_0098_beckhoff.TcDUT
{attribute 'pack_mode' := '1'} //Ensures 1-byte-alignmend
TYPE AX5000_P_0098_beckhoff :
STRUCT
	Actual_lenght : UINT := 16#80;
	Max_lenght : UINT := 16#80;
	Name_plate_type: E_AX5000_P_0150_DigitalNamePlate;
//	{attribute 'hide'}
	Rsvd1:ARRAY[0..0] OF UINT;
	Id_prat_1:UDINT;
	Id_prat_2:UDINT;
	Version_no:UINT;
	Motor_vendor:UINT;
	Serial_number:UDINT;
	Motor_type:STRING(29);
	Feedback_typ:STRING(29);
//	{attribute 'hide'}
	Rsvd2:UINT;
	Add_motor_parameter_description:UINT;
	Nominal_current:UDINT;
	Nominal_voltage:UINT;
	Nominal_frequenz:UINT;
	Nominal_speed:UINT;
	Maximun_speed:UINT;
	Cos_phi:UINT;
	Maximum_feedback_speed:UINT;
//	{attribute 'hide'}
	Rsvd3:ARRAY[0..5] OF UINT;	
//	{attribute 'hide'}
	Rsvd4:UINT;
	Checksum:UINT;
	Position_offset:UDINT;
	Number_of_adjustments:UINT;
	
	Additional_mech_position_offset:UDINT;
	Checksum2:UINT;
(*
	Vendor:STRING(29);
	Order_code:STRING(29);
	Electric_type:STRING(29);
	Serial_no:STRING(10);
	 {attribute 'hide'}
	rsvd5:ARRAY[0..9] OF UINT;
	Mechanical_commutation_offset:UDINT;
	Generic:ARRAY[0..61] OF UINT;*)
END_STRUCT
END_TYPE

// ---- POUs/IO/Drives/SoE/Ax5000ParamSTRUCTs/P/AX5000_P_0098_beckhoff_electrical_data.TcDUT
{attribute 'pack_mode' := '1'}//Ensures 1-byte-alignmend
TYPE AX5000_P_0098_beckhoff_electrical_data :
STRUCT
	Actual_lenght:UINT;
	Max_lenght:UINT;
	Name_plate_type:UINT;
//	 {attribute 'hide'}
	Rsvd1:ARRAY[0..0] OF UINT;
	(*Id_prat_1:UDINT;
	Id_prat_2:UDINT;
	Version_no:UINT;
	Motor_vendor:UINT;
	Serial_number:UDINT;
	Motor_type:STRING(29);
	Feedback_typ:STRING(29);
	 {attribute 'hide'}
	rsvd2:UINT;
	Add_motor_parameter_description:UINT;
	Nominal_current:UDINT;
	Nominal_voltage:UINT;
	Nominal_frequenz:UINT;
	Nominal_speed:UINT;
	Maximun_speed:UINT;
	Cos_phi:UINT;
	Maximum_feedback_speed:UINT;
	 {attribute 'hide'}
	Rsvd3:ARRAY[0..5] OF UINT;
	Checksum:UINT;
	Position_offset:UDINT;
	Number_of_adjustments:UINT;
	Additional_mech_position_offset:UDINT;
	Checksum2:UINT;*)

	Vendor:STRING(29);
	Order_code:STRING(29);
	Electric_type:STRING(29);
	Serial_no:STRING(9);
//	{attribute 'hide'}
	Rsvd5:ARRAY[0..9] OF UINT;
	Mechanical_commutation_offset:UDINT;
	(*Generic:ARRAY[0..61] OF UINT;*)
END_STRUCT
END_TYPE

// ---- POUs/IO/Drives/SoE/Ax5000ParamSTRUCTs/P/AX5000_P_0099.TcDUT
{attribute 'pack_mode' := '1'}//Ensures 1-byte-alignmend
TYPE AX5000_P_0099 :
STRUCT
	Actual_lenght:UINT;
	Max_lenght:UINT;
	Request:UINT;
	Encoder_connector:UINT;
	File:UINT;
	File_size_in_words:UINT;
//	{attribute 'hide'}
	Rsvd:ARRAY [0..1] OF UINT;
	Offset_in_Words:UINT;
	Length_in_words:UINT;
	Response:UINT;
	Data_state:UINT;
	File_size_in_words2:UINT;
//	{attribute 'hide'}
	Rsvd1:UINT;
//	{attribute 'hide'}
	Rsvd2: UDINT;
	Offset_in_words2:UINT;
	Length_in_words2:UINT;
	Data_array:ARRAY[0..255] OF UINT;

END_STRUCT
END_TYPE

// ---- POUs/IO/Drives/SoE/Ax5000ParamSTRUCTs/P/AX5000_P_0100.TcDUT
TYPE AX5000_P_0100 :
STRUCT
	ASM_nominal_speed:UDINT;
END_STRUCT
END_TYPE

// ---- POUs/IO/Drives/SoE/Ax5000ParamSTRUCTs/P/AX5000_P_0103.TcDUT
TYPE AX5000_P_0103 :
STRUCT
	ASM_boost_voltage:UINT;
END_STRUCT
END_TYPE

// ---- POUs/IO/Drives/SoE/Ax5000ParamSTRUCTs/P/AX5000_P_0105.TcDUT
TYPE AX5000_P_0105 :
STRUCT
	ASM_Rotor_time_constant:UINT;
END_STRUCT
END_TYPE

// ---- POUs/IO/Drives/SoE/Ax5000ParamSTRUCTs/P/AX5000_P_0107.TcDUT
TYPE AX5000_P_0107 :
STRUCT
	ASM_Magnetizing_current:UDINT;
END_STRUCT
END_TYPE

// ---- POUs/IO/Drives/SoE/Ax5000ParamSTRUCTs/P/AX5000_P_0109.TcDUT
TYPE AX5000_P_0109 :
STRUCT
	ASM_stator_leakage_inductance:UDINT;
END_STRUCT
END_TYPE

// ---- POUs/IO/Drives/SoE/Ax5000ParamSTRUCTs/P/AX5000_P_0111.TcDUT
TYPE AX5000_P_0111 :
STRUCT
	ASM_rotor_leakage_inductance:UDINT;
END_STRUCT
END_TYPE

// ---- POUs/IO/Drives/SoE/Ax5000ParamSTRUCTs/P/AX5000_P_0112.TcDUT
TYPE AX5000_P_0112 :
STRUCT
	ASM_acceleration_control_torque_limit_value:UINT;
END_STRUCT
END_TYPE

// ---- POUs/IO/Drives/SoE/Ax5000ParamSTRUCTs/P/AX5000_P_0115.TcDUT
TYPE AX5000_P_0115 :
STRUCT
	ASM_stall_protection_loop_torque_limit_value:UINT;
END_STRUCT
END_TYPE

// ---- POUs/IO/Drives/SoE/Ax5000ParamSTRUCTs/P/AX5000_P_0117.TcDUT
TYPE AX5000_P_0117 :
STRUCT
	ASM_stall_protection_loop_intrgral_action_time:UINT;
END_STRUCT
END_TYPE

// ---- POUs/IO/Drives/SoE/Ax5000ParamSTRUCTs/P/AX5000_P_0151.TcDUT
{attribute 'pack_mode' := '1'}//Ensures 1-byte-alignmend
TYPE AX5000_P_0151 :
STRUCT
	Actual_lenght:UINT;
	Max_lenght:UINT;
	Manufacturer:UINT;
	Feedback_type:UINT;
	Feedback_type_string:STRING(29);
//{attribute 'hide'}
	Rsvd1:ARRAY[0..4] OF UINT;
	Process_channel:ARRAY[0..11] OF UINT;
	Parameter_channel:ARRAY[0..77] OF UINT;
	Manufacturer_limits_settings:ARRAY[0..5] OF UINT;
//{attribute 'hide'}
	Rsvd2:ARRAY[0..7] OF UINT;
END_STRUCT
END_TYPE

// ---- POUs/IO/Drives/SoE/Ax5000ParamSTRUCTs/P/AX5000_P_0153.TcDUT
TYPE AX5000_P_0153 :
STRUCT
	Feedback_1_geat_denominator:UDINT;
END_STRUCT
END_TYPE

// ---- POUs/IO/Drives/SoE/Ax5000ParamSTRUCTs/P/AX5000_P_0155.TcDUT
TYPE AX5000_P_0155 :
STRUCT
	Feedback_1_resolution_scaling:UDINT;
END_STRUCT
END_TYPE

// ---- POUs/IO/Drives/SoE/Ax5000ParamSTRUCTs/P/AX5000_P_0165.TcDUT
{attribute 'pack_mode' := '1'}//Ensures 1-byte-alignmend
TYPE AX5000_P_0165 :
STRUCT
	Actual_lenght:UINT;
	Max_lenght:UINT;
	Command_mode:UINT;
	Activation:UINT;
	
//{attribute 'hide'}
	Rsvd1:ARRAY[0..1] OF UINT;
	Current_level:UINT;
	Duration:UINT;
//{attribute 'hide'}
	Rsvd2:ARRAY[0..3] OF UINT;
	First_phase_current_level:UINT;
	First_phase_ramp_up_time:UINT;
	Second_phase_current_level:UINT;
	Second_phase_ramp_up_time:UINT;
	Commutation_pos_control_Kp:UINT;
	First_phase_pos_monitoring_limit:UINT;
	First_phase_step_width:UINT;
	First_phase_wating_time_after_step:UINT;
	Second_phase_duration:UINT;
	Error_monitoring:UINT;
//{attribute 'hide'}
	Rsvd3:ARRAY[0..9] OF UINT;


END_STRUCT
END_TYPE

// ---- POUs/IO/Drives/SoE/Ax5000ParamSTRUCTs/P/AX5000_P_0167.TcDUT
{attribute 'pack_mode' := '1'}//Ensures 1-byte-alignmend
TYPE AX5000_P_0167 :
STRUCT
	Actual_lenght:UINT;
	Max_lenght:UINT;
	eMode:UINT;
	Current_level:UINT;
	Moving_distance:UINT;
	Velocety:UINT;
//{attribute 'hide'}
	Rsvd:UINT;
//{attribute 'hide'}
	Rsvd2:UINT;
	EqualDirektions:UINT;
	Commutation_position_difference:UINT;
//{attribute 'hide'}
	Rsvd3:UINT;
//{attribute 'hide'}
	Rsvd4:UINT;

END_STRUCT
END_TYPE

// ---- POUs/IO/Drives/SoE/Ax5000ParamSTRUCTs/P/AX5000_P_0168.TcDUT
{attribute 'pack_mode' := '1'}//Ensures 1-byte-alignmend
TYPE AX5000_P_0168 :
STRUCT
	Actual_lenght:UINT;
	Max_lenght:UINT;
	Phase_shift:UINT;
	Sin_offset_correction:UINT;
	Cos_offset_correction:UINT;
//{attribute 'hide'}
	Rsvd:ARRAY[0..6] OF UINT;
	Vector_length:UINT;
	Sin_max:UINT;
	Sin_min:UINT;
	Cos_max:UINT;
	Cos_min:UINT;
//{attribute 'hide'}
	Rsvd2:ARRAY[0..4] OF UINT;

END_STRUCT
END_TYPE

// ---- POUs/IO/Drives/SoE/Ax5000ParamSTRUCTs/P/AX5000_P_0171.TcDUT
{attribute 'pack_mode' := '1'}//Ensures 1-byte-alignmend
TYPE AX5000_P_0171 :
STRUCT
	Actual_lenght:UINT;
	Max_lenght:UINT;
	Numeration:UDINT;
	Denominator:UDINT;
	Mask:UDINT;
	Position_offset:UDINT;
	Data_valid:UINT;
//{attribute 'hide'}
	Rsvd:UINT;
END_STRUCT
END_TYPE

// ---- POUs/IO/Drives/SoE/Ax5000ParamSTRUCTs/P/AX5000_P_0182.TcDUT
TYPE AX5000_P_0182 :
STRUCT
	Feedback_2_geat_numerator:UDINT;
END_STRUCT
END_TYPE

// ---- POUs/IO/Drives/SoE/Ax5000ParamSTRUCTs/P/AX5000_P_0185.TcDUT
TYPE AX5000_P_0185 :
STRUCT
	Feedback_2_resolution_scaling:UDINT;
END_STRUCT
END_TYPE

// ---- POUs/IO/Drives/SoE/Ax5000ParamSTRUCTs/P/AX5000_P_0192.TcDUT
TYPE AX5000_P_0192 :
STRUCT
	Feedback2_save_digital_nameplate:UINT;
END_STRUCT
END_TYPE

// ---- POUs/IO/Drives/SoE/Ax5000ParamSTRUCTs/P/AX5000_P_0193.TcDUT
TYPE AX5000_P_0193 :
STRUCT
	Scan_feedback2:UINT;
END_STRUCT
END_TYPE

// ---- POUs/IO/Drives/SoE/Ax5000ParamSTRUCTs/P/AX5000_P_0199.TcDUT
TYPE AX5000_P_0199 :
STRUCT
	Direct_feedback_access:UINT;
END_STRUCT
END_TYPE

// ---- POUs/IO/Drives/SoE/Ax5000ParamSTRUCTs/P/AX5000_P_0216.TcDUT
TYPE AX5000_P_0216 :
STRUCT
	Max_DC_Link_voltage:UINT;
END_STRUCT
END_TYPE

// ---- POUs/IO/Drives/SoE/Ax5000ParamSTRUCTs/P/AX5000_P_0218.TcDUT
TYPE AX5000_P_0218 :
STRUCT
	Internal_brake_resistor_actual_peak_energy:UINT;
END_STRUCT
END_TYPE

// ---- POUs/IO/Drives/SoE/Ax5000ParamSTRUCTs/P/AX5000_P_0221.TcDUT
{attribute 'pack_mode' := '1'}//Ensures 1-byte-alignmend
TYPE AX5000_P_0221 :
STRUCT
	Actual_lenght:UINT;
	Max_lenght:UINT;
	Max_energy_over_100percent_duty_cycle:UDINT;
	Max_energy_over_40percent_duty_cycle:UDINT;
	Max_energy_over_20percent_duty_cycle:UDINT;
	Max_energy_over_10percent_duty_cycle:UDINT;
	Max_energy_over_1percent_duty_cycle:UDINT;
	Max_energy_over_01percent_duty_cycle:UDINT;
END_STRUCT
END_TYPE

// ---- POUs/IO/Drives/SoE/Ax5000ParamSTRUCTs/P/AX5000_P_0250.TcDUT
TYPE AX5000_P_0250 :
STRUCT
	Scource:UINT;
END_STRUCT
END_TYPE

// ---- POUs/IO/Drives/SoE/Ax5000ParamSTRUCTs/P/AX5000_P_0271.TcDUT
TYPE AX5000_P_0271 :
STRUCT
	Save_sosition_offset_pc:UINT;
END_STRUCT
END_TYPE

// ---- POUs/IO/Drives/SoE/Ax5000ParamSTRUCTs/P/AX5000_P_0272.TcDUT
{attribute 'pack_mode' := '1'}//Ensures 1-byte-alignmend
TYPE AX5000_P_0272 :
STRUCT
	Actual_Length : UINT := 8;
	Max_Length : UINT := 8;
	(* FeedbackNumber &amp; MemorySelection *)
	Data : BYTE;
//	{attribute 'hide'}
	Rsvd1 : ARRAY [1..3] OF USINT;
	Position_Offset : UDINT;	
END_STRUCT
END_TYPE

// ---- POUs/IO/Drives/SoE/Ax5000ParamSTRUCTs/P/AX5000_P_0277.TcDUT
TYPE AX5000_P_0277 :
STRUCT
	Schedule_modulo_init_data_saving:UINT;
END_STRUCT
END_TYPE

// ---- POUs/IO/Drives/SoE/Ax5000ParamSTRUCTs/P/AX5000_P_0278.TcDUT
TYPE AX5000_P_0278 :
STRUCT
	Ignore_for_one_PreOp_SafeOp_transition:UINT;
END_STRUCT
END_TYPE

// ---- POUs/IO/Drives/SoE/Ax5000ParamSTRUCTs/P/AX5000_P_0300.TcDUT
TYPE AX5000_P_0300 :
STRUCT
	Actual_lenght:UINT;
	Max_lenght:UINT;
	Error_number_history:ARRAY[0..99] OF UDINT;
END_STRUCT
END_TYPE

// ---- POUs/IO/Drives/SoE/Ax5000ParamSTRUCTs/P/AX5000_P_0306.TcDUT
TYPE AX5000_P_0306 :
STRUCT
	Actual_main_loop_time:UINT;
END_STRUCT
END_TYPE

// ---- POUs/IO/Drives/SoE/Ax5000ParamSTRUCTs/P/AX5000_P_0307.TcDUT
TYPE AX5000_P_0307 :
STRUCT
	Max_main_loop_time:UINT;
END_STRUCT
END_TYPE

// ---- POUs/IO/Drives/SoE/Ax5000ParamSTRUCTs/P/AX5000_P_0309.TcDUT
TYPE AX5000_P_0309 :
STRUCT
	Max_ctrl_loop_time:UINT;
END_STRUCT
END_TYPE

// ---- POUs/IO/Drives/SoE/Ax5000ParamSTRUCTs/P/AX5000_P_0317.TcDUT
TYPE AX5000_P_0317 :
STRUCT
	Actual_amplifier_stilisation:UDINT;
END_STRUCT
END_TYPE

// ---- POUs/IO/Drives/SoE/Ax5000ParamSTRUCTs/P/AX5000_P_0321.TcDUT
{attribute 'pack_mode' := '1'}
TYPE AX5000_P_0321 :
STRUCT
	Actual_lenght:UINT;
	Max_lenght:UINT;
	Disc_size:UDINT;
	Usend_size:UDINT;
	Alignment:UDINT;
	Free_size:UDINT;
(*File 0*)
	Type0:UINT;
//	{attribute 'hide'}
	rsvd0:UINT;
	Version0:UINT;
	Build0:UINT;
	Time_H0:UDINT;
	Time_L0:UDINT;
	Id10:UINT;
	Id20:UINT;
	Size0:UDINT;
	Size_on_disk0:UDINT;
	alignment0:UDINT;
	Start_adresse0:UDINT;

(*File 1*)
	Type1:UINT;
//	{attribute 'hide'}
	Rsvd1:UINT;
	Version1:UINT;
	Build1:UINT;
	Time_H1:UDINT;
	Time_L1:UDINT;
	Id11:UINT;
	Id21:UINT;
	Size1:UDINT;
	Size_on_disk1:UDINT;
	alignment1:UDINT;
	Start_adresse1:UDINT;

(*File 2*)
	Type2:UINT;
//	{attribute 'hide'}
	Rsvd2:UINT;
	Version2:UINT;
	Build2:UINT;
	Time_H2:UDINT;
	Time_L2:UDINT;
	Id12:UINT;
	Id22:UINT;
	Size2:UDINT;
	Size_on_disk2:UDINT;
	alignment2:UDINT;
	Start_adresse2:UDINT;

(*File 3*)
	Type3:UINT;
//	{attribute 'hide'}
	Rsvd3:UINT;
	Version3:UINT;
	Build3:UINT;
	Time_H3:UDINT;
	Time_L3:UDINT;
	Id13:UINT;
	Id23:UINT;
	Size3:UDINT;
	Size_on_disk3:UDINT;
	alignment3:UDINT;
	Start_adresse3:UDINT;

(*File 4*)
	Type4:UINT;
//	{attribute 'hide'}
	Rsvd4:UINT;
	Version4:UINT;
	Build4:UINT;
	Time_H4:UDINT;
	Time_L4:UDINT;
	Id14:UINT;
	Id24:UINT;
	Size4:UDINT;
	Size_on_disk4:UDINT;
	alignment4:UDINT;
	Start_adresse4:UDINT;

(*File 5*)
	Type5:UINT;
//	{attribute 'hide'}
	Rsvd5:UINT;
	Version5:UINT;
	Build5:UINT;
	Time_H5:UDINT;
	Time_L5:UDINT;
	Id15:UINT;
	Id25:UINT;
	Size5:UDINT;
	Size_on_disk5:UDINT;
	alignment5:UDINT;
	Start_adresse5:UDINT;

(*File 6*)
	Type6:UINT;
//	{attribute 'hide'}
	Rsvd6:UINT;
	Version6:UINT;
	Build6:UINT;
	Time_H6:UDINT;
	Time_L6:UDINT;
	Id16:UINT;
	Id26:UINT;
	Size6:UDINT;
	Size_on_disk6:UDINT;
	alignment6:UDINT;
	Start_adresse6:UDINT;

(*File 7*)
	Type7:UINT;
//	{attribute 'hide'}
	Rsvd7:UINT;
	Version7:UINT;
	Build7:UINT;
	Time_H7:UDINT;
	Time_L7:UDINT;
	Id17:UINT;
	Id27:UINT;
	Size7:UDINT;
	Size_on_disk7:UDINT;
	Alignment7:UDINT;
	Start_adresse7:UDINT;

(*File 8*)
	Type8:UINT;
//	{attribute 'hide'}
	Rsvd8:UINT;
	Version8:UINT;
	Build8:UINT;
	Time_H8:UDINT;
	Time_L8:UDINT;
	Id18:UINT;
	Id28:UINT;
	Size8:UDINT;
	Size_on_disk8:UDINT;
	Alignment8:UDINT;
	Start_adresse8:UDINT;

(*File 9*)
	Type9:UINT;
	Rsvd9:UINT;
	Version9:UINT;
	Build9:UINT;
	Time_H9:UDINT;
	Time_L9:UDINT;
	Id19:UINT;
	Id29:UINT;
	Size9:UDINT;
	Size_on_disk9:UDINT;
	alignment9:UDINT;
	Start_adresse9:UDINT;
END_STRUCT
END_TYPE

// ---- POUs/IO/Drives/SoE/Ax5000ParamSTRUCTs/P/AX5000_P_0322.TcDUT
//	{attribute 'hide'}
TYPE AX5000_P_0322 :
STRUCT
	Actual_lenght:UINT;
	Max_lenght:UINT;


	PCB_ID_version:UINT;
	Hwld1:UINT;
	Hwld2:UINT;
	Hwld3:UINT;
	Manufacturing_Data:UINT;
	Serial_number_low:UINT;
	Serial_number_high:UINT;
	Checksum:UINT;


	PCB_ID_version1:UINT;
	Hwld4:UINT;
	Hwld5:UINT;
	Hwld6:UINT;
	Manufacturing_Data1:UINT;
	Serial_number_low1:UINT;
	Serial_number_high1:UINT;
	Checksum1:UINT;


	PCB_ID_version2:UINT;
	Hwld7:UINT;
	Hwld8:UINT;
	Hwld9:UINT;
	Manufacturing_Data2:UINT;
	Serial_number_low2:UINT;
	Serial_number_high2:UINT;
	Checksum2:UINT;


	PCB_ID_version3:UINT;
	Hwld10:UINT;
	Hwld11:UINT;
	Hwld12:UINT;
	Manufacturing_Data3:UINT;
	Serial_number_low3:UINT;
	Serial_number_high3:UINT;
	Checksum3:UINT;


	PCB_ID_version4:UINT;
	Hwld13:UINT;
	Hwld14:UINT;
	Hwld15:UINT;
	Manufacturing_Data4:UINT;
	Serial_number_low4:UINT;
	Serial_number_high4:UINT;
	Checksum4:UINT;


	PCB_ID_version5:UINT;
	Hwld16:UINT;
	Hwld17:UINT;
	Hwld18:UINT;
	Manufacturing_Data5:UINT;
	Serial_number_low5:UINT;
	Serial_number_high5:UINT;
	Checksum5:UINT;


	Control_Pcb_Id_valid:UINT;
	Power_Pcb_Id_valid:UINT;
	Driver_Pcb_Id_valid:UINT;
	Front_Pcb_Id_valid:UINT;
	OptionSlot_Pcb_Id_valid:UINT;
	SafetySlot_Id_valid:UINT;
	Dsp_Revidion:UINT;
	Dsp_Id_Xint_Revision:UINT;
	Feedback_Dsp_Id:UINT;
	Feedback_Dsp_Revision:UINT;
	Esc_Revision:UINT;
	Esc_build:UINT;
	Esc_type:UINT;
	FPGA_device_Type:UINT;
	FPGA_device_Subtype:UINT;
	FPGA_version_number:UINT;
	FPGA_build_number:UINT;
	Option_slot_FPGA:UINT;
END_STRUCT
END_TYPE

// ---- POUs/IO/Drives/SoE/Ax5000ParamSTRUCTs/P/AX5000_P_0326.TcDUT
TYPE AX5000_P_0326 :
STRUCT
	Actual_lenght:UINT;
	Max_lenght:UINT;
	Release_note:STRING;
END_STRUCT
END_TYPE

// ---- POUs/IO/Drives/SoE/Ax5000ParamSTRUCTs/P/AX5000_P_0353.TcDUT
TYPE AX5000_P_0353 :
STRUCT
	Emergency_stop_jerk:UDINT;
END_STRUCT
END_TYPE

// ---- POUs/IO/Drives/SoE/Ax5000ParamSTRUCTs/P/AX5000_P_0361.TcDUT
TYPE AX5000_P_0361 :
STRUCT
	Actual_lenght:UINT;
	Max_lenght:UINT;
	Parameter_set_configuration:ARRAY[0..34] OF UINT;
END_STRUCT
END_TYPE

// ---- POUs/IO/Drives/SoE/Ax5000ParamSTRUCTs/P/AX5000_P_0400.TcDUT
TYPE AX5000_P_0400 EXTENDS ST_AX5000_P_0400:
STRUCT
//	Hardware_enable_configuration:UINT;
END_STRUCT
END_TYPE

// ---- POUs/IO/Drives/SoE/Ax5000ParamSTRUCTs/P/AX5000_P_0401.TcDUT
TYPE AX5000_P_0401 :
STRUCT
	Positiv_limit_switch: ST_AX5000_P_0401_LimitSwitch;
	Negativ_limit_switch: ST_AX5000_P_0401_LimitSwitch;
END_STRUCT
END_TYPE

// ---- POUs/IO/Drives/SoE/Ax5000ParamSTRUCTs/P/AX5000_P_0452.TcDUT
TYPE AX5000_P_0452 :
STRUCT
	Current_controller_control_word:UINT;
END_STRUCT
END_TYPE

// ---- POUs/IO/Drives/SoE/Ax5000ParamSTRUCTs/P/AX5000_P_0453.TcDUT
TYPE AX5000_P_0453 :
STRUCT
	Current_controller_status_word:UINT;
END_STRUCT
END_TYPE

// ---- POUs/IO/Drives/SoE/Ax5000ParamSTRUCTs/P/AX5000_P_0455.TcDUT
{attribute 'pack_mode' := '1'}
TYPE AX5000_P_0455 :
STRUCT
	Actual_lenght:UINT;
	Max_lenght:UINT;
	Mode:UINT;
	Rsvd:UINT;
	Min_voltage:UINT;
	Max_voltage:UINT;
	Max_current_for_fielweakening:UDINT;
	Max_velocity_for_fielweakening:UDINT;
END_STRUCT
END_TYPE

// ---- POUs/IO/Drives/SoE/Ax5000ParamSTRUCTs/P/AX5000_P_0460.TcDUT
TYPE AX5000_P_0460 :
STRUCT
	Actual_flux_generating_current:UINT;
END_STRUCT
END_TYPE

// ---- POUs/IO/Drives/SoE/Ax5000ParamSTRUCTs/P/AX5000_P_0462.TcDUT
TYPE AX5000_P_0462 :
STRUCT
	Actual_peak_current_limit:UINT;
END_STRUCT
END_TYPE

// ---- POUs/IO/Drives/SoE/Ax5000ParamSTRUCTs/P/AX5000_P_0463.TcDUT
TYPE AX5000_P_0463 :
STRUCT
	Actual_current_limit:UINT;
END_STRUCT
END_TYPE

// ---- POUs/IO/Drives/SoE/Ax5000ParamSTRUCTs/P/AX5000_P_0502.TcDUT
TYPE AX5000_P_0502 :
STRUCT
	Velocity_controller_control_word:UINT;
END_STRUCT
END_TYPE

// ---- POUs/IO/Drives/SoE/Ax5000ParamSTRUCTs/P/AX5000_P_0513.TcDUT
{attribute 'pack_mode' := '1'}
TYPE AX5000_P_0513 :
STRUCT
	Actual_lenght:UINT;
	Max_lenght:UINT;
	ST_CONV_Version:UINT;
	Rsvd1:UINT;
	Filter_type:UINT;
//	{attribute 'hide'}
	nRsvd2:UINT;
	Low_pass_frequency:UDINT;
	Low_pass_damping:UDINT;
	High_pass_frequency:UDINT;
	High_pass_damping:UDINT;
//	{attribute 'hide'}
	Rsvd3:UDINT;
//	{attribute 'hide'}
	Rsvd4:UDINT;
	QMath_factor:UINT;
//	{attribute 'hide'}
	nRsvd5:UINT;
	b0:UDINT;
	b1:UDINT;
	b2:UDINT;
	a1:UDINT;
	a2:UDINT;
//	{attribute 'hide'}
	Rsvd6:UDINT;
	Rsvd7:UDINT;
END_STRUCT
END_TYPE

// ---- POUs/IO/Drives/SoE/Ax5000ParamSTRUCTs/P/AX5000_P_0552.TcDUT
TYPE AX5000_P_0552 :
STRUCT
	Position_controller_word:UINT;
END_STRUCT
END_TYPE

// ---- POUs/IO/Drives/SoE/Ax5000ParamSTRUCTs/P/AX5000_P_0555.TcDUT
TYPE AX5000_P_0555 :
STRUCT
	Position_command_value_monitoring_window:UINT;
END_STRUCT
END_TYPE

// ---- POUs/IO/Drives/SoE/Ax5000ParamSTRUCTs/P/AX5000_P_0558.TcDUT
TYPE AX5000_P_0558 :
STRUCT
	Position_controller_output:DINT;
END_STRUCT
END_TYPE

// ---- POUs/IO/Drives/SoE/Ax5000ParamSTRUCTs/P/AX5000_P_0611.TcDUT
TYPE AX5000_P_0611 :
STRUCT
	Configurable_status_word:UINT;
END_STRUCT
END_TYPE

// ---- POUs/IO/Drives/SoE/Ax5000ParamSTRUCTs/P/AX5000_P_0802.TcDUT
TYPE AX5000_P_0802 :
STRUCT
	Digital_output:UINT;
END_STRUCT
END_TYPE

// ---- POUs/IO/Drives/SoE/Ax5000ParamSTRUCTs/P/AX5000_P_0810.TcDUT
TYPE AX5000_P_0810 :
STRUCT
	Actual_lenght:UINT;
	Max_lenght:UINT;
	Funktion_number:UDINT;
	Code_word:UDINT;
	Parameter1:UDINT;
	Parameter2:UDINT;
	Parameter3:UDINT;
	Parameter4:UDINT;
	Parameter5:UDINT;

END_STRUCT
END_TYPE

// ---- POUs/IO/Drives/SoE/Ax5000ParamSTRUCTs/P/AX5000_P_0901.TcDUT
TYPE AX5000_P_0901 :
STRUCT
	Safe_factory_settings:UINT;
END_STRUCT
END_TYPE

// ---- POUs/IO/Drives/SoE/Ax5000ParamSTRUCTs/P/AX5000_P_0904.TcDUT
TYPE AX5000_P_0904 :
STRUCT
	Save_device_component_hardware_Ids:UINT;
END_STRUCT
END_TYPE

// ---- POUs/IO/Drives/SoE/Ax5000ParamSTRUCTs/P/AX5000_P_0906.TcDUT
TYPE AX5000_P_0906 :
STRUCT
	Reset_operation_times:UINT;
END_STRUCT
END_TYPE

// ---- POUs/IO/Drives/SoE/Ax5000ParamSTRUCTs/P/AX5000_P_1002.TcDUT
TYPE AX5000_P_1002 :
STRUCT
	Debug_pointer_1_value:UDINT;
END_STRUCT
END_TYPE

// ---- POUs/IO/Drives/SoE/Ax5000ParamSTRUCTs/P/AX5000_P_1003.TcDUT
TYPE AX5000_P_1003 :
STRUCT
	Debug_pointer_2_adr:UDINT;
END_STRUCT
END_TYPE

// ---- POUs/IO/Drives/SoE/Ax5000ParamSTRUCTs/P/AX5000_P_1005.TcDUT
TYPE AX5000_P_1005 :
STRUCT
	Debug_pointer_2_value:UDINT;
END_STRUCT
END_TYPE

// ---- POUs/IO/Drives/SoE/Ax5000ParamSTRUCTs/P/AX5000_P_1006.TcDUT
TYPE AX5000_P_1006 :
STRUCT
	Addr:UINT;
	Source:UINT;
END_STRUCT
END_TYPE

// ---- POUs/IO/Drives/SoE/Ax5000ParamSTRUCTs/P/AX5000_P_1011.TcDUT
TYPE AX5000_P_1011 :
STRUCT
	Feedback_debug_pointer_2_value:UINT;
END_STRUCT
END_TYPE

// ---- POUs/IO/Drives/SoE/Ax5000ParamSTRUCTs/P/AX5000_P_1012.TcDUT
TYPE AX5000_P_1012 :
STRUCT
	Memory_dump_selector:UINT;
END_STRUCT
END_TYPE

// ---- POUs/IO/Drives/SoE/Ax5000ParamSTRUCTs/P/AX5000_P_1020.TcDUT
TYPE AX5000_P_1020 :
STRUCT
	Debug_parameter:UINT;
END_STRUCT
END_TYPE

// ---- POUs/IO/Drives/SoE/Ax5000ParamSTRUCTs/P/AX5000_P_1021.TcDUT
TYPE AX5000_P_1021 :
STRUCT
	Debug_variable:UDINT;
END_STRUCT
END_TYPE

// ---- POUs/IO/Drives/SoE/Ax5000ParamSTRUCTs/S/AX5000_S_0002.TcDUT
TYPE AX5000_S_0002 :
STRUCT
	Communication_cycle_time:UINT;
END_STRUCT
END_TYPE

// ---- POUs/IO/Drives/SoE/Ax5000ParamSTRUCTs/S/AX5000_S_0012.TcDUT
TYPE AX5000_S_0012 :
STRUCT
	Class_2_diagnostic:UINT;
END_STRUCT
END_TYPE

// ---- POUs/IO/Drives/SoE/Ax5000ParamSTRUCTs/S/AX5000_S_0017.TcDUT
TYPE AX5000_S_0017 :
STRUCT
	Actual_lenght:UINT;
	Max_lenght:UINT;
	IDN_list_of_all_operation_data: ARRAY[0..693] OF UINT;
END_STRUCT
END_TYPE

// ---- POUs/IO/Drives/SoE/Ax5000ParamSTRUCTs/S/AX5000_S_0033.TcDUT
TYPE AX5000_S_0033 :
STRUCT
	Secondary_operation_mode1:UINT;
END_STRUCT
END_TYPE

// ---- POUs/IO/Drives/SoE/Ax5000ParamSTRUCTs/S/AX5000_S_0034.TcDUT
TYPE AX5000_S_0034 :
STRUCT
	Secondary_operation_mode2:UINT;
END_STRUCT
END_TYPE

// ---- POUs/IO/Drives/SoE/Ax5000ParamSTRUCTs/S/AX5000_S_0040.TcDUT
TYPE AX5000_S_0040 :
STRUCT
	Velocity_feedback_value1:DINT;
END_STRUCT
END_TYPE

// ---- POUs/IO/Drives/SoE/Ax5000ParamSTRUCTs/S/AX5000_S_0043.TcDUT
TYPE AX5000_S_0043 :
STRUCT
	Velocity_polarity_parameter:UINT;
END_STRUCT
END_TYPE

// ---- POUs/IO/Drives/SoE/Ax5000ParamSTRUCTs/S/AX5000_S_0044.TcDUT
TYPE AX5000_S_0044 :
STRUCT
	Velocity_data_scaling_type:UINT;
END_STRUCT
END_TYPE

// ---- POUs/IO/Drives/SoE/Ax5000ParamSTRUCTs/S/AX5000_S_0045.TcDUT
TYPE AX5000_S_0045 :
STRUCT
	Velocity_data_scaling_factor:UINT;
END_STRUCT
END_TYPE

// ---- POUs/IO/Drives/SoE/Ax5000ParamSTRUCTs/S/AX5000_S_0046.TcDUT
TYPE AX5000_S_0046 :
STRUCT
	Velocity_data_scaling_exponent:INT;
END_STRUCT
END_TYPE

// ---- POUs/IO/Drives/SoE/Ax5000ParamSTRUCTs/S/AX5000_S_0047.TcDUT
TYPE AX5000_S_0047 :
STRUCT
	Position_command_valut:DINT;
END_STRUCT
END_TYPE

// ---- POUs/IO/Drives/SoE/Ax5000ParamSTRUCTs/S/AX5000_S_0079.TcDUT
TYPE AX5000_S_0079 :
STRUCT
	Rotational_position_resolution:UDINT;
END_STRUCT
END_TYPE

// ---- POUs/IO/Drives/SoE/Ax5000ParamSTRUCTs/S/AX5000_S_0084.TcDUT
TYPE AX5000_S_0084 :
STRUCT
	Torque_feedback_value:INT;
END_STRUCT
END_TYPE

// ---- POUs/IO/Drives/SoE/Ax5000ParamSTRUCTs/S/AX5000_S_0085.TcDUT
TYPE AX5000_S_0085 EXTENDS ST_AX5000_S_0085:
STRUCT
//	Torque_polarity_parameter:UINT;
END_STRUCT
END_TYPE

// ---- POUs/IO/Drives/SoE/Ax5000ParamSTRUCTs/S/AX5000_S_0103.TcDUT
TYPE AX5000_S_0103 :
STRUCT
	Moduo_value:UDINT;
END_STRUCT
END_TYPE

// ---- POUs/IO/Drives/SoE/Ax5000ParamSTRUCTs/S/AX5000_S_0107.TcDUT
TYPE AX5000_S_0107 :
STRUCT
	Current_conrol_loop_integral_action_time1:UINT;
END_STRUCT
END_TYPE

// ---- POUs/IO/Drives/SoE/Ax5000ParamSTRUCTs/S/AX5000_S_0113.TcDUT
TYPE AX5000_S_0113 :
STRUCT
	Maximum_motor_speed:UDINT;
END_STRUCT
END_TYPE

// ---- POUs/IO/Drives/SoE/Ax5000ParamSTRUCTs/S/AX5000_S_0130.TcDUT
TYPE AX5000_S_0130 :
STRUCT
	Probe_value_1_positive_edge:DINT;
END_STRUCT
END_TYPE

// ---- POUs/IO/Drives/SoE/Ax5000ParamSTRUCTs/S/AX5000_S_0169.TcDUT
TYPE AX5000_S_0169 :
STRUCT
//	Probe_control_parameter:UINT;
	
(* 0=Not Active, 1=Active *)
		Probe1PositiveEdge : BIT;
		(* 0=Not Active, 1=Active *)
		Probe1NegativeEdge : BIT;
		 {attribute 'hide'}
		_reserved1 : BIT;
		 {attribute 'hide'}
		_reserved2 : BIT;
		 {attribute 'hide'}
		_reserved3 : BIT;
		(* 0=Single Measuring, 1=Continous Measuring *)
		ModeProbe1 : BIT;
		 {attribute 'hide'}
		_reserved4 : BIT;
		 {attribute 'hide'}
		_reserved5 : BIT;
		(* 0=Ativation with S170, 1=Autoactivation from SafeOp to Op *)
		AutoActivation : BIT;
		 {attribute 'hide'}
		_reserved6 : BIT;
		 {attribute 'hide'}
		_reserved7 : BIT;
		 {attribute 'hide'}
		_reserved8 : BIT;
		 {attribute 'hide'}
		_reserved9 : BIT;
		 {attribute 'hide'}
		_reserved10 : BIT;
		 {attribute 'hide'}
		_reserved11 : BIT;
		 {attribute 'hide'}
		_reserved12 : BIT;
END_STRUCT
END_TYPE

// ---- POUs/IO/Drives/SoE/Ax5000ParamSTRUCTs/S/AX5000_S_0170.TcDUT
TYPE AX5000_S_0170 :
STRUCT
	Probing_cycle_procedure_command:UINT;
END_STRUCT
END_TYPE

// ---- POUs/IO/Drives/SoE/Ax5000ParamSTRUCTs/S/AX5000_S_0186.TcDUT
TYPE AX5000_S_0186 :
STRUCT
	Length_of_the_configurabel_data_record_in_the_MDT:UINT;
END_STRUCT
END_TYPE

// ---- POUs/IO/Drives/SoE/Ax5000ParamSTRUCTs/S/AX5000_S_0196.TcDUT
TYPE AX5000_S_0196 :
STRUCT
	Motor_rated_current:UDINT;
END_STRUCT
END_TYPE

// ---- POUs/IO/Drives/SoE/Ax5000ParamSTRUCTs/S/AX5000_S_0203.TcDUT
TYPE AX5000_S_0203 :
STRUCT
	Amplifier_shut_down_temperature:UINT;
END_STRUCT
END_TYPE

// ---- POUs/IO/Drives/SoE/Ax5000ParamSTRUCTs/S/AX5000_S_0204.TcDUT
TYPE AX5000_S_0204 :
STRUCT
	Motor_shut_down_temperature:UINT;
END_STRUCT
END_TYPE

// ---- POUs/IO/Drives/SoE/Ax5000ParamSTRUCTs/S/AX5000_S_0206.TcDUT
TYPE AX5000_S_0206 :
STRUCT
	Drive_of_delay_time:UINT;
END_STRUCT
END_TYPE

// ---- POUs/IO/Drives/SoE/Ax5000ParamSTRUCTs/S/AX5000_S_0207.TcDUT
TYPE AX5000_S_0207 :
STRUCT
	Drive_delay_time:UINT;
END_STRUCT
END_TYPE

// ---- POUs/IO/Drives/SoE/Ax5000ParamSTRUCTs/S/AX5000_S_0273.TcDUT
TYPE AX5000_S_0273 :
STRUCT
	Maximum_drive_off_delay_time:UDINT;
END_STRUCT
END_TYPE

// ---- POUs/IO/Drives/SoE/Ax5000ParamSTRUCTs/S/AX5000_S_0381.TcDUT
TYPE AX5000_S_0381 :
STRUCT
	DC_bus_current:DINT;
END_STRUCT
END_TYPE

// ---- POUs/IO/Drives/SoE/Ax5000ParamSTRUCTs/S/AX5000_S_0403.TcDUT
TYPE AX5000_S_0403 :
STRUCT
	Position_feedback_value_status:UINT;
END_STRUCT
END_TYPE

// ---- POUs/IO/Drives/SoE/Ax5000ParamSTRUCTs/S/AX5000_S_0405.TcDUT
TYPE AX5000_S_0405 :
STRUCT
	Probe1_enable:UINT;
END_STRUCT
END_TYPE

// ---- POUs/IO/Drives/SoE/Ax5000ParamSTRUCTs/S/AX5000_S_0432.TcDUT
TYPE AX5000_S_0432 :
STRUCT
	Actual_lenght:UINT;
	Max_lenght:UINT;
	Serial_number_drive_control:STRING(18);
END_STRUCT
END_TYPE

// ---- POUs/IO/Drives/SoE/Ax5000ParamSTRUCTs/S/AX5000_S_0436.TcDUT
TYPE AX5000_S_0436 :
STRUCT
	Operating_time_power_stage:UDINT;
END_STRUCT
END_TYPE

// ---- POUs/_Miscellaneous/TC_VN_COLORS.TcDUT
TYPE TC_VN_COLORS :
STRUCT
	// Colors
	BLACK		: TcVnVector4_LREAL := [0, 0, 0, 255];
	WHITE		: TcVnVector4_LREAL := [255, 255, 255, 255];
	RED			: TcVnVector4_LREAL := [255, 0, 0, 255];
	LIME		: TcVnVector4_LREAL := [0, 255, 0, 255]; //bright green
	BLUE		: TcVnVector4_LREAL := [0, 0, 255, 255];
	YELLOW		: TcVnVector4_LREAL := [255, 255, 0, 255];
	CYAN		: TcVnVector4_LREAL := [0, 255, 255, 255];	
	MAGENTA		: TcVnVector4_LREAL := [255, 0, 255, 255];
	SILVER		: TcVnVector4_LREAL := [192,192,192, 255];
	GRAY		: TcVnVector4_LREAL := [128,128,128, 255]; //darker than silver
	MAROON		: TcVnVector4_LREAL := [128,0,0, 255];
	OLIVE		: TcVnVector4_LREAL := [128,128,0, 255];
	GREEN		: TcVnVector4_LREAL := [0,128,0, 255]; //darker green
	PURPLE		: TcVnVector4_LREAL := [128,0,128, 255];
	TEAL		: TcVnVector4_LREAL := [0,128,128, 255];
	NAVY		: TcVnVector4_LREAL := [0,0,128, 255];
END_STRUCT
END_TYPE

// ---- POUs/_Miscellaneous/COLOR.TcDUT
TYPE COLOR :
STRUCT
	NULL									: UDINT := 16#00000000;
	BLACK									: UDINT := 16#FF000000;	
	YELLOW									: UDINT := 16#FFFFFF00;
	RED										: UDINT := 16#FFFF0000;
	BLUE									: UDINT := 16#FF0000FF;
	GREEN									: UDINT := 16#FF008000;
	GREY									: UDINT := 16#FF808080;
	GREYDARK								: UDINT := 16#FFC0C0C0;
	PINK									: UDINT := 16#FFFFC0CB;
	ORANGE									: UDINT := 16#FFFFA500;
	VIOLET									: UDINT := 16#FFEE82EE;
	WHITE									: UDINT := 16#FFFFFFFF;																										
END_STRUCT
END_TYPE

// ---- POUs/_Miscellaneous/LCID.TcDUT
{attribute 'qualified_only'}
TYPE LCID :
STRUCT
// Code: 	https://de.wikipedia.org/wiki/ISO-3166-1-Kodierliste
// LCID:	https://msdn.microsoft.com/de-de/goglobal/bb964664.aspx
// LCID:	https://winprotocoldoc.blob.core.windows.net/productionwindowsarchives/MS-LCID/%5bMS-LCID%5d.pdf

//	ISO3166 ALPHA-2, ALPHA-3
	NONE						: eLCID := eLCID.NONE;
	CZ,CZE						: eLCID := eLCID.CZ; // Czech - 1029 
	DK,DNK						: eLCID := eLCID.DK; // Danish - 1030
	DE,DEU						: eLCID := eLCID.DE; // German - 1033	
	GR,GRC						: eLCID := eLCID.GR; // Greek - 1032
	US,USA						: eLCID := eLCID.US; // English(US) - 1033
	ES,ESP						: eLCID := eLCID.ES; // Spainsh(Spain) - 1034
	FI,FIN						: eLCID := eLCID.FI; // Finnish - 1035
	FR,FRA						: eLCID := eLCID.FR; // French(France) - 1036	
	IT,ITA						: eLCID := eLCID.IT; // Italian - 1040
	NL,NLD						: eLCID := eLCID.NL; // Dutch(Netherlands) - 1043
	NO,NOR						: eLCID := eLCID.NO; // Norwegian - 1044
	PL,POL						: eLCID := eLCID.PL; // Polish - 1045
	RU,RUS						: eLCID := eLCID.RU; // Russian - 1049
	SE,SWE						: eLCID := eLCID.SE; // Swedish(Sweden) - 1053
	CA,CAN						: eLCID := eLCID.CA; // Canadian - 1099
	TR,TUR						: eLCID := eLCID.TR; // Turkish - 1055
	CN,CHN						: eLCID := eLCID.CN; // Chinese(CN-Simplified) - 2052
	GB,GBR						: eLCID := eLCID.GB; // English(UK) - 2057	
	PT,PRT						: eLCID := eLCID.PT; // Portuguese(Portugal) - 2057	
END_STRUCT
END_TYPE

// ---- POUs/Safety/SAFETY_CIRCUIT_STATUS.TcDUT
TYPE SAFETY_CIRCUIT_STATUS :
STRUCT
	State													:	eSTATE := eSTATE.ABORTED;

	InAborting												:	BOOL; //MonOut switched to false, MonDelOut still true
	InAborted												:	BOOL; //MonOut and MonDelOut = FALSE
	InClearing												:	BOOL; //MonOut and MonDelOut = TRUE, OK delay time is running
	InIdle													:	BOOL; //OK = TRUE
	OK														:	BOOL; //On/Off Delay Signal
	OK_2													:	BOOL; //On/Off Delay Signal 2 - between OK and MonDelOut delay time
	RT														:	BOOL; //R trig based on OK
	FT														:	BOOL; //F trig based on MonDelOut
                            								
//Hardwaresignal       								
	ReadyToRestart											:	BOOL := FALSE; //TRUE when restart of safety circuit is executable 
	MonOut													:	BOOL := FALSE; //output
	MonDelOut												:	BOOL := FALSE; //output delayed
END_STRUCT
END_TYPE

// ---- Version/Global_Version.TcGVL
{attribute 'TcGenerated'}
{attribute 'no-analysis'}
{attribute 'linkalways'}
// This function has been automatically generated from the project information.
VAR_GLOBAL CONSTANT
	{attribute 'const_non_replaced'}
	stLibVersion_EngineeringToolbox : ST_LibVersion := (iMajor := 3, iMinor := 1, iBuild := 2, iRevision := 4, nFlags := 0, sVersion := '3.1.2.4');
END_VAR

// ---- POUs/IO/Cylinder/I_Cylinder.TcIO
INTERFACE I_Cylinder EXTENDS I_ActuatorWorkBase

METHOD enable : BOOL //Result value = successful execution of desired action 
VAR_INPUT
	IN							:	BOOL; //TRUE = to Work pos / FLASE = to base pos
END_VAR
END_METHOD

{attribute 'monitoring' := 'call'}
PROPERTY PUBLIC inError : Bool
GET
END_GET
END_PROPERTY

{attribute 'monitoring' := 'call'}
PROPERTY isBusy : BOOL
GET
END_GET
END_PROPERTY

{attribute 'monitoring' := 'call'}
PROPERTY isInBasePos : BOOL
GET
END_GET
END_PROPERTY

{attribute 'monitoring' := 'call'}
PROPERTY isInWorkPos : BOOL
GET
END_GET
END_PROPERTY

METHOD PUBLIC moveToBasePos : BOOL //Return = Done -> InBasePos
END_METHOD

METHOD PUBLIC moveToWorkPos : BOOL //Return = Done -> InWorkPos
END_METHOD

{attribute 'monitoring' := 'call'}
PROPERTY noFeed : BOOL
GET
END_GET
END_PROPERTY

{attribute 'monitoring' := 'call'}
PROPERTY PUBLIC rCylinder : REFERENCE TO Cylinder
GET
END_GET
END_PROPERTY

{attribute 'monitoring' := 'call'}
PROPERTY simulation : BOOL
GET
END_GET
SET
END_SET
END_PROPERTY

METHOD PUBLIC switchOff : BOOL
VAR_INPUT
END_VAR
END_METHOD

END_INTERFACE

// ---- POUs/IO/_ItfActuators/I_ActuatorBase.TcIO
INTERFACE I_ActuatorBase EXTENDS __System.IQueryInterface

{attribute 'monitoring' := 'call'}
PROPERTY public inError : bool
GET
END_GET
END_PROPERTY

{attribute 'monitoring' := 'call'}
PROPERTY public isBusy : bool
GET
END_GET
END_PROPERTY

{attribute 'monitoring' := 'call'}
PROPERTY public isOff : BOOL
GET
END_GET
END_PROPERTY

{attribute 'monitoring' := 'call'}
PROPERTY public noFeed : BOOL
GET
END_GET
END_PROPERTY

{attribute 'monitoring' := 'call'}
PROPERTY public ok : bool
GET
END_GET
END_PROPERTY

METHOD PUBLIC reset : BOOL
VAR_INPUT
END_VAR
END_METHOD

METHOD public switchOff : BOOL
VAR_INPUT
END_VAR
END_METHOD

END_INTERFACE

// ---- POUs/IO/_ItfActuators/I_ActuatorEnableDisable.TcIO
INTERFACE I_ActuatorEnableDisable EXTENDS I_ActuatorBase

{attribute 'monitoring' := 'call'}
PROPERTY public isDisabled : BOOL
GET
END_GET
END_PROPERTY

{attribute 'monitoring' := 'call'}
PROPERTY public isEnabled : BOOL
GET
END_GET
END_PROPERTY

METHOD public setDisable : BOOL
VAR_INPUT
END_VAR
END_METHOD

METHOD public setEnable : BOOL
VAR_INPUT
END_VAR
END_METHOD

END_INTERFACE

// ---- POUs/IO/_ItfActuators/I_ActuatorOpenClose.TcIO
INTERFACE I_ActuatorOpenClose EXTENDS I_ActuatorBase

{attribute 'monitoring' := 'call'}
PROPERTY public isClosed : BOOL
GET
END_GET
END_PROPERTY

{attribute 'monitoring' := 'call'}
PROPERTY public isOpened : BOOL
GET
END_GET
END_PROPERTY

METHOD public setClose : BOOL
VAR_INPUT
END_VAR
END_METHOD

METHOD public setOpen : BOOL
VAR_INPUT
END_VAR
END_METHOD

END_INTERFACE

// ---- POUs/IO/_ItfActuators/I_ActuatorWorkBase.TcIO
INTERFACE I_ActuatorWorkBase EXTENDS I_ActuatorBase

{attribute 'monitoring' := 'call'}
PROPERTY isInBasePos : BOOL
GET
END_GET
END_PROPERTY

{attribute 'monitoring' := 'call'}
PROPERTY isInWorkPos : BOOL
GET
END_GET
END_PROPERTY

METHOD public moveToBasePos : BOOL
VAR_INPUT
END_VAR
END_METHOD

METHOD public moveToWorkPos : BOOL
VAR_INPUT
END_VAR
END_METHOD

END_INTERFACE

// ---- POUs/Motion/TF50xx-NC/00_Base/I_AxNcPTP.TcIO
INTERFACE I_AxNcPTP EXTENDS I_AxNcBase

{attribute 'monitoring' := 'call'}
PROPERTY rMotion : REFERENCE TO AxMotion
GET
END_GET
END_PROPERTY

END_INTERFACE

// ---- POUs/Connectivity/TF6340-SerialCom/ComPortDeviceCom/ComPortDeviceCom_SendRecString.TcPOU
//FB sends a "command" out and waits for response of the connected device (handshake mode)
//By changing the Fnc the FB mode can be switched into only send or only receive
FUNCTION_BLOCK ComPortDeviceCom_SendRecString
VAR CONSTANT
	TIMEOUT_COM												: TIME 		:= T#10S;
END_VAR
VAR_OUTPUT CONSTANT
	FNC_SEND_REC											:	INT := 0; //Send command and wait for response
	FNC_SEND												:	INT := 1; //Send only
	FNC_REC													:	INT := 2; //Receive only
END_VAR
VAR_INPUT
	Execute													: BOOL;
	Fnc														:	INT(FNC_SEND_REC..FNC_SEND_REC) := FNC_SEND_REC;
	ClrComBuffer											: BOOL; //TRUE Clears com buffer before start
	RecTimeout												: TIME := DEFAULT_ADS_TIMEOUT; 
	Command													: T_MAxSTRing;	//Suffix will be added
	Prefix													: STRING(5) := '';
	Suffix													: STRING(5) := '$r$n';  //Will be addet to send data and removed from response
END_VAR
VAR_IN_OUT
	Handle													:	ComPortDeviceCom_BufferHandle;
END_VAR
VAR_OUTPUT
	ResponseLen												: UDINT;
	Response												: T_MaxString;
	Done													: BOOL;
	Busy													: BOOL;
	Error													: BOOL;
	ErrorID													: ComError_t := ComError_t.COMERROR_NOERROR;
END_VAR
VAR
(* Memory *****************************************************)
	state													: INT := 0;
	
(* Timer ******************************************************)
	timeout													:	ton := (PT := TIMEOUT_COM);
(* Trigger ****************************************************)
	rtExecute												: R_TRIG;
	
(* Blocks *****************************************************)
	Rec														: ReceiveString255 := (Timeout := T#10S);
	Send													: SendString255;
	
(* Error ******************************************************)
(* Dummys *****************************************************)
END_VAR

	(* Send text and receive response						 *)
	(*********************************************************)
	
(* state machine ********************************************************)
	rtExecute(CLK := Execute);
	CASE state OF
	0 : 
		Busy 												:= FALSE;
		IF NOT Execute THEN
			Done 											:= FALSE;
			Error 											:= FALSE;
			ErrorID 										:= 0;
		END_IF
		IF rtExecute.Q THEN
			Busy 											:= TRUE;		
			timeout(IN := FALSE, PT := TIMEOUT_COM + RecTimeout);
			ResponseLen 									:= 0;
			Error 											:= FALSE;
			ErrorID 										:= ComError_t.COMERROR_NOERROR;
			Rec(Reset := TRUE,Timeout := RecTimeout, rxBuffer := Handle.RxBUffer , ReceivedString := Response, Prefix := Prefix, Suffix := Suffix  );
			
			IF ClrComBuffer
			THEN
				handle.Clear();
			END_IF
			
			IF Fnc = FNC_REC
			THEN //only receive 
				MemSet(ADR(Response),0,SIZEOF(Response));
				Rec(Reset := FALSE, rxBuffer := handle.RxBUffer , ReceivedString := Response );
				State										:= 2;				
			ELSE
				Send(SendString := CONCAT(Command, Suffix),TxBuffer := Handle.TXBuffer);	
				state 										:= state + 1;
			END_IF
				
		END_IF
		
	1 : //Send tag 
		IF Send.Busy 
		THEN  //Call FB only if still busy after call in state 0
			Send(SendString := CONCAT(Command, Suffix),TxBuffer := handle.TxBuffer); 
		END_IF
		IF NOT Send.Busy 
		THEN
			IF Send.Error <> ComError_t.COMERROR_NOERROR
			THEN
				Busy										:= FALSE;
				Error										:= TRUE;
				Errorid										:= Send.Error;
				state										:= 0;
			ELSIF Fnc = FNC_SEND
			THEN
				Busy										:= FALSE;
				Done										:= TRUE;
				state										:= 0;				
			ELSE
				MemSet(ADR(Response),0,SIZEOF(Response));
				Rec(Reset := FALSE, rxBuffer := handle.RxBUffer , ReceivedString := Response );
				state 										:= state + 1;
			END_IF
		END_IF

	2: //Wair for response
		timeout(IN := TRUE);
		Rec(ReceivedString	:= Response,RXbuffer := Handle.RxBuffer);	
		IF NOT Rec.Busy
		THEN
			IF Rec.StringReceived
			THEN
				IF LEN(Response) > 0
				THEN
					IF Suffix[0] <> 0 //Cut suffix if selected 
					THEN
						Response							:= ReadStrToSeperator(Suffix,Response);
					END_IF
					ResponseLen								:= TO_UDINT(LEN(Response));	
					Busy									:= FALSE;
					Done									:= TRUE;
					state									:= 0;	
				ELSE
					; //Nothing received, continue to read until done or timeout kicks in
				END_IF
				
			ELSIF Rec.Error <> ComError_t.COMERROR_NOERROR
			THEN
				Busy										:= FALSE;
				Error										:= TRUE;
				Errorid										:= Rec.Error;
				state										:= 0;					
					
			ELSIF Rec.RxTimeout
			THEN
				Busy										:= FALSE;
				Error										:= TRUE;
				Errorid										:= ComError_t.COMERROR_TIMEOUT;
				state										:= 0;	
			ELSIF timeout.Q
			THEN
				Busy										:= FALSE;
				Error										:= TRUE;
				Errorid										:= ComError_t.COMERROR_TIMEOUT;
				state										:= 0;					
			END_IF
		END_IF
	END_CASE
(********************************************************************************)

END_FUNCTION_BLOCK

// ---- POUs/Connectivity/TF6340-SerialCom/ComPortBasic/ComPortBackground.TcPOU
{attribute 'no_check'}
//Wrapper for background communication of serial com ports like EL terminal or PC-COM-Port
//based on TF6340 - SerialCommunication (Tc2_SerialCom)
FUNCTION_BLOCK ComPortBackground
VAR_INPUT
	Enable													: BOOL ; // FB will be processed as long as enable is TRUE 
	ResetTrig												: BOOL ; // The function block will be reset with a rising edge 
	Mode													: ComSerialLineMode_t := SERIALLINEMODE_EL6_22B; //terminal parameter, see ComSerialLineMode_t at documentation of library
	pComIn													: POINTER TO BYTE;	// COM-Port process image	%I*
	pComOut													: POINTER TO BYTE;	// COM-Port process image  	%Q* 
	SizeComIn												: UINT := 22; 	// Size of process data - depends on terminal type (3,5,22,64 Byte)
	Cfg 													: ComSerialConfig := (Baudrate := 19200); // Cfg Structure for PC-com port
	TXBuffer												: COMbuffer ;	// TX buffer used by ComPortSendRec
END_VAR
VAR_OUTPUT
	RXBuffer												: COMbuffer ;	// RX buffer used by ComPortSendRec
	PortOpened												: BOOL;	// Background communication etablished
	Busy													: BOOL;	// Busy is TRUE at the rising edge of Enable and stays TRUE as long as the FB is performing any action. 
	Error													: BOOL; // Rising edge of Error informs that an error occurred during the execution of the Function Block 
{attribute 'displaymode':='hex'}
	ErrorId													: UDINT;// Error identification - see ADS return codes and TF6340 documentation at Beckhoff infosys for further information
	ComErrorId												: ComError_t ; 	// Serial com. error indentification - Tc2_SerialCom documentaion for further information
END_VAR
VAR_IN_OUT
END_VAR
VAR
(* internally used variables ********************************************************)
	MemErrorID												: UDINT := 0;
	State													: INT := 0;
	
(* internal function-block instances for serial communication ***************************************************************)
	_ClearComBuffer											: 	ClearComBuffer; // clears the internal communication buffer of the PLC
	_SerLineControl											: 	SerialLineControl; // looks after backround-communication
	_SerLineControlADS										: 	SerialLineControlADS; // looks after backround-communication
	_Comreset												: 	ComReset; // Reset KL-Terminal

END_VAR

(*******************************************************************************)

CASE state OF
0:
	IF NOT Enable AND NOT _SerLineControlADS.Busy
		OR Error
	THEN
		Busy												:= FALSE;
		PortOpened											:= FALSE;
		
		IF ResetTrig
		THEN
			reset();
		END_IF

	ELSIF Mode = ComSerialLineMode_t.SERIALLINEMODE_PC_COM_PORT
	THEN
		_SerLineControlADS(	Connect		:= Enable,
							SerialCfg	:= Cfg,
							NetId		:= '',
							Timeout		:= ,
							TxBuffer	:= TXBuffer,
							RxBuffer	:= RXBuffer,
							PortOpened	=> PortOpened,
							Error		=> ,
							ErrorID		=> ,
							Busy		=> ,
							TxBufCount	=> ,
							RxBufCount	=> );
		
		Busy 												:= TRUE;

		IF _SerLineControlADS.Error 
		THEN
			Error											:= TRUE;
			ErrorId											:= _SerLineControlAds.ErrorId;
//			ComErrorId										:= _SerLineControlAds.ErrorId; // missing cast !
		END_IF

	ELSIF Enable
	THEN
		_SerLineControl(
			Mode		:= mode ,
			pComIn		:= pComIn ,
			pComOut		:= pComOut ,
			SizeComIn	:= UINT_TO_INT(SizeComIn),
			TxBuffer	:= TXBuffer ,
			RxBuffer	:= RXBuffer ,
			Error		=> ,
			ErrorID		=> );
		
		Busy												:= TRUE;

		IF _SerLineControl.Error 
		THEN
			Error											:= TRUE;
			ErrorId											:= TO_UDINT(_SerLineControl.ErrorId);
			ComErrorId										:= _SerLineControl.ErrorId;
		ELSE
			PortOpened										:= TRUE;
		END_IF
	END_IF

20: (* Reset ******************************************)
	_ComReset(	Execute		:= FALSE,
				pComIn		:= pComIn,
				pComOut		:= pComOut ,
				SizeComIn	:= SizeComIn ,
				Done		=> ,
				Busy		=> ,
				Error		=> ,
				ErrorID		=> );

	(* Buffer leeren *)
	_ClearComBuffer(Buffer:= TXBuffer);
	_ClearComBuffer(Buffer:= RXBuffer);

	state 													:= 21;

21:
	_ComReset(	Execute		:= Mode <> ComSerialLineMode_t.SERIALLINEMODE_PC_COM_PORT,
				pComIn		:= pComIn,
				pComOut		:= pComOut ,
				SizeComIn	:= SizeComIn ,
				Done		=> ,
				Busy		=> ,
				Error		=> ,
				ErrorID		=> );
										
	IF NOT _ComReset.Busy
	THEN
		IF _ComReset.Error
		THEN
			Error											:= TRUE;
			ErrorId											:= INT_TO_UDINT(_ComReset.ErrorID);
			ComErrorId										:= _ComReset.ErrorID;
		END_IF
		_ComReset(Execute := FALSE, pComIn	:= pComIn, pComOut := pComOut , SizeComIn := SizeComIn);
		State 												:= SEL(Mode = ComSerialLineMode_t.SERIALLINEMODE_PC_COM_PORT, 0, 90);
	END_IF

90: (* Error ******************************************)
	_SerLineControlADS(	Connect		:= FALSE,
						SerialCfg	:= Cfg,
						NetId		:= '',
						Timeout		:= ,
						TxBuffer	:= TXBuffer,
						RxBuffer	:= RXBuffer,
						PortOpened	=> PortOpened,
						Error		=> ,
						ErrorID		=> ,
						Busy		=> ,
						TxBufCount	=> ,
						RxBufCount	=> );

	IF NOT _SerLineControlADS.Busy
	THEN
		PortOpened											:= FALSE;
		Busy												:= FALSE;
		state												:= 0;
	END_IF
	
END_CASE


(***********************************************************************************************)

METHOD PUBLIC reset : BOOL //Return value = TRUE if execution finished
VAR_INPUT
END_VAR
IF Error OR NOT Enable
THEN //jump to reset state
	state 													:= SEL(state < 20 OR state > 21 ,state , 20);
	Error													:= FALSE;
	ErrorId													:= 0;
	ComErrorId												:= ComError_t.COMERROR_NOERROR;
	reset													:= TRUE;
ELSE
	reset													:= FALSE;
END_IF
END_METHOD

END_FUNCTION_BLOCK

// ---- POUs/Connectivity/TF6340-SerialCom/ComPortDeviceCom/ComPortEL6x22BEasyConnect.TcPOU
//FB handles the backround communication to an EL6xxx in 22byte mode via FB  ComPortBackground and provides and handle to be used for FBs DeviceCom_SendRecBytes/String
FUNCTION_BLOCK ComPortEL6x22BEasyConnect
VAR_INPUT
	Enable													: BOOL; 
	Reset													: BOOL; //Calls ComReset FB
	ComOut											AT %Q*	:	EL6OutData22B;
END_VAR		
VAR_IN_OUT
	
END_VAR
VAR_OUTPUT
	Connected												: BOOL;
	ComIn											AT %I*	:	EL6inData22B;
	Handle													:	ComPortDeviceCom_BufferHandle;
	Error													: BOOL;
	{attribute 'displaymode':='hex'}  
	ErrorId													: ComError_t;
END_VAR

VAR
(*  Memory *****************************************************)
	
(*  Timer ******************************************************)

(*  Trigger ****************************************************)

(*  Blocks *****************************************************)
	ComBackground		 									:	ComPortBackground;
END_VAR
	
VAR CONSTANT
END_VAR

ComBackground(
	Enable		:= Enable, 
	ResetTrig	:= Reset, 
	Mode		:= SERIALLINEMODE_EL6_22B, 
	pComIn		:= ADR(ComIn), 
	pComOut		:= ADR(ComOut), 
	SizeComIn	:= SIZEOF(ComIn), 
	Cfg			:= , 
	TXBuffer	:= Handle.TXBuffer, 
	RXBuffer	=> Handle.RXBuffer, 
	PortOpened	=> Connected, 
	Busy		=> , 
	Error		=> Error, 
	ErrorId		=> , 
	ComErrorId	=> ErrorId);

METHOD PUBLIC reset : BOOL
VAR_INPUT
END_VAR
reset := ComBackground.reset();
IF reset THEN Handle.Clear(); END_IF
END_METHOD

END_FUNCTION_BLOCK

// ---- POUs/Connectivity/TF625x-Modbus/Master/TF6250-ModbusTcpServer/TCP/ModbusTcpMaster.TcPOU
{attribute 'no_check'}
// ModBus comunication master to multible slaves useing TCP protocol	
// based on TF6250 - required lib: Tc2_ModbusTCP
FUNCTION_BLOCK ModbusTcpMaster
VAR_OUTPUT CONSTANT
	MIN_SLAVE												:	INT := 1;
	MAX_SLAVE												:	INT := PARAM.MODBUS_MAX_SLAVES_OF_MASTER;
{attribute 'displaymode':='binary'}
	OPTION_DISABLE_ERROR_STATE								:	BYTE := 2#0000_0001; //FB will not go into error state and keeps running, even all slaves are in error state
END_VAR
VAR_INPUT
	Enable													:	BOOL ; 	// FB will be processed as long as enable is TRUE 
	ResetTrig												:	BOOL ; 	// The function block will be reset with a rising edge 
{attribute 'displaymode':='binary'}
	Options													:	BYTE := 0; //FB options, see VAR_OUTPUT CONSTANT
	SlaveCom												:	ARRAY[MIN_SLAVE..MAX_SLAVE] OF POINTER TO ModbusSlaveCom;
	Timestamp												:	DT;
END_VAR         	
VAR_OUTPUT      	
	JobNo													:	INT := 0;
	SlaveNo													:	INT := 0;
{attribute 'displaymode':='binary'}
	SlaveInErrorMask										:	DWORD; //Bit.1 indicates slave 1 in error
	Error													:	BOOL; 	// Rising edge of Error informs that an error occurred during the execution of the Function Block 
{attribute 'displaymode':='hex'}
	ErrorID													:	UDINT; 	// Error identification - see ADS return codes at Beckhoff infosys for further information 
	ErrorText												:	STRING;
END_VAR
VAR
(* memory **************************************************)
	state 													:	INT := 0;

(* trigger *************************************************)

(* timer ***************************************************)

(* blocks **************************************************)
	ReadCoils												:	FB_MBReadCoils := (tTimeout	 := DEFAULT_ADS_TIMEOUT);			// Fnc 1
	ReadInputs												:	FB_MBReadInputs := (tTimeout := DEFAULT_ADS_TIMEOUT);			// Fnc 2
	ReadRegs												:	FB_MBReadRegs := (tTimeout	:= DEFAULT_ADS_TIMEOUT);			// Fnc 3
	ReadInputRegs											:	FB_MBReadInputRegs := (tTimeout	:= DEFAULT_ADS_TIMEOUT);		// Fnc 4
	WriteSingleCoil											:	FB_MBWriteSingleCoil := (tTimeout	:= DEFAULT_ADS_TIMEOUT);	// Fnc 5
	WriteSingleReg											:	FB_MBWriteSingleReg := (tTimeout:= DEFAULT_ADS_TIMEOUT);		// Fnc 6
	Diagnose												:	FB_MBDiagnose := (tTimeout	:= DEFAULT_ADS_TIMEOUT);			// Fnc 8
	WriteCoils												:	FB_MBWriteCoils := (tTimeout:= DEFAULT_ADS_TIMEOUT);			// Fnc 15
	WriteRegs												:	FB_MBWriteRegs := (tTimeout	:= DEFAULT_ADS_TIMEOUT);			// Fnc 16
	ReadWriteRegs											:	FB_MBReadWriteRegs := (tTimeout	:= DEFAULT_ADS_TIMEOUT); 		// Fnc 23	use read and write job instead
(* internal used variables *********************************)
	i,j,k													:	INT :=0;
END_VAR

	IF ResetTrig THEN
		reset();
	END_IF
		
	CASE state OF
	0:	(* Idle *)
		IF Enable 
		THEN
			k 												:=	0;
			JobNo  :=  SlaveNo								:=	1;
			state 											:=	10;
		END_IF

	10: 
		IF GetNextSlave() 
		THEN (* find Slave *)
			k 												:= 0;
			IF GetNextJob() 
			THEN (* find JobNo *)
				SlaveCom[SlaveNo]^.currentJobIdx 			:= JobNo;
				SlaveCom[SlaveNo]^.writeJobRequested 		:= SlaveCom[SlaveNo]^.Jobs[JobNo].FunctionCode >= 5;
				State 										:= SEL(SlaveCom[SlaveNo]^.writeJobRequested, 20, 15);
			END_IF
		ELSE
			state 											:=	0;
		END_IF
			
	15: (* wait for valid write date *)
		IF NOT SlaveCom[SlaveNo]^.writeJobRequested
		THEN
			SlaveCom[SlaveNo]^.Jobs[JobNo].Valid 			:= FALSE;
			state 											:= 20;
		END_IF

	20: (* start job *)	
		IF NOT StartJob(FALSE) // Not Busy,Execute set to false
		THEN						
			state 											:= 30;
		END_IF

	30: (* wait for com cycle *)
		IF NOT StartJob(TRUE) THEN // Not Busy, Execute set to True
			IF Error
			THEN
				ErrorText									:= CONCAT('Error at SlaveNo: ',	CONCAT(INT_TO_STRING(SlaveNo), CONCAT(', JobNo: ', INT_TO_STRING(JobNo))));
				SlaveCom[SlaveNo]^.countBad 				:= SlaveCom[SlaveNo]^.countBad +1;
				SlaveInErrorMask							:= CSETBIT32(SlaveInErrorMask,TO_SINT(SlaveNo),TRUE);
				IF Options.0
				THEN
					JobNo 									:= JobNo + 1;
					state 									:= 10;	(* next job *)				
				ELSE
					state 									:= 98; 					
				END_IF
			ELSE
				SlaveInErrorMask							:= CSETBIT32(SlaveInErrorMask,TO_SINT(SlaveNo),FALSE);
				SlaveCom[SlaveNo]^.countGood 				:= SlaveCom[SlaveNo]^.countGood +1;
				SlaveCom[SlaveNo]^.Jobs[JobNo].Valid 		:= TRUE;
				SlaveCom[SlaveNo]^.Jobs[JobNo].TimeStamp 	:= Timestamp;
				JobNo 										:= JobNo + 1;
				state 										:= 10;	(* next job *)
			END_IF
			StartJob(FALSE);
		END_IF

	98: (* wait for quit *)
		;

	END_CASE

METHOD PRIVATE getNextJob : Bool //Return value = TRUE if execution finished
VAR_INPUT
END_VAR
	
	WHILE SlaveCom[SlaveNo]^.Jobs[JobNo].FunctionCode = 0 DO
		JobNo 											:= JobNo + 1;
		IF JobNo > SlaveCom[SlaveNo]^.MAX_SLAVE_JOB THEN
			JobNo 										:= SlaveCom[SlaveNo]^.MIN_SLAVE_JOB;
			SlaveNo 									:= SlaveNo + 1;
			GetNextJob									:= FALSE;
			RETURN;
		END_IF
	END_WHILE
	GetNextJob											:= TRUE;
END_METHOD

METHOD PRIVATE getNextSlave : Bool //Return value = TRUE if execution finished
VAR_INPUT
END_VAR
	WHILE SlaveCom[SlaveNo] = 0 OR_ELSE NOT SlaveCom[SlaveNo]^.Enable DO
		SlaveNo 										:= SlaveNo + 1;
		IF SlaveNo > MAX_SLAVE 
		THEN
			k 											:= k + 1;
			SlaveNo 									:= MIN_SLAVE;
		ELSIF k = 2 
		THEN
			k 											:= 0;
			GetNextSlave								:= FALSE;
			RETURN;
		END_IF	
	END_WHILE
	GetNextSlave										:= TRUE;
END_METHOD

METHOD PUBLIC reset : bool //Return value = TRUE if execution finished
VAR_INPUT
END_VAR
IF State = 98 
THEN
	state													:= 0;
END_IF
Error														:= FALSE;
ErrorID														:= 0;
ErrorText													:= '';
reset														:= TRUE;
END_METHOD

METHOD PRIVATE startJob : BOOL //Return value = TRUE as long as the job is busy
VAR_INPUT
	Execute							: BOOL;
END_VAR
	IF 	SlaveCom[SlaveNo]^.Jobs[JobNo].FunctionCode = 1 THEN
		ReadCoils(
			sIPAddr			:= SlaveCom[SlaveNo]^.ipAddr, 
			nTCPPort		:= TO_UINT(SlaveCom[SlaveNo]^.Port), 
			nUnitID			:= SlaveCom[SlaveNo]^.Address, 
			nQuantity		:= SlaveCom[SlaveNo]^.jobs[JobNo].Quantity, 
			nMBAddr			:= SlaveCom[SlaveNo]^.jobs[JobNo].startAddress, 
			cbLength		:= SlaveCom[SlaveNo]^.jobs[JobNo].Quantity, 
			pDestAddr		:= ADR(SlaveCom[SlaveNo]^.Data), 
			bExecute		:= Execute, 
			tTimeout		:= , 
			bBusy			=> StartJob, 
			bError			=> Error, 
			nErrId			=> ErrorID);
			
	ELSIF 	SlaveCom[SlaveNo]^.Jobs[JobNo].FunctionCode = 2 THEN
		ReadInputs(
			sIPAddr			:= SlaveCom[SlaveNo]^.ipAddr, 
			nTCPPort		:= TO_UINT(SlaveCom[SlaveNo]^.Port), 
			nUnitID			:= SlaveCom[SlaveNo]^.Address, 
			nQuantity		:= SlaveCom[SlaveNo]^.jobs[JobNo].Quantity, 
			nMBAddr			:= SlaveCom[SlaveNo]^.jobs[JobNo].startAddress, 
			cbLength		:= SlaveCom[SlaveNo]^.jobs[JobNo].Quantity, 
			pDestAddr		:= ADR(SlaveCom[SlaveNo]^.Data), 
			bExecute		:= Execute, 
			tTimeout		:= , 
			bBusy			=> StartJob, 
			bError			=> Error, 
			nErrId			=> ErrorID);
			
	ELSIF 	SlaveCom[SlaveNo]^.Jobs[JobNo].FunctionCode = 3 THEN
		ReadRegs(
			sIPAddr			:= SlaveCom[SlaveNo]^.ipAddr, 
			nTCPPort		:= TO_UINT(SlaveCom[SlaveNo]^.Port), 
			nUnitID			:= SlaveCom[SlaveNo]^.Address, 
			nQuantity		:= SlaveCom[SlaveNo]^.jobs[JobNo].Quantity, 
			nMBAddr			:= SlaveCom[SlaveNo]^.jobs[JobNo].startAddress, 
			cbLength		:= SlaveCom[SlaveNo]^.jobs[JobNo].Quantity * 2, 
			pDestAddr		:= ADR(SlaveCom[SlaveNo]^.Data), 
			bExecute		:= Execute, 
			tTimeout		:= , 
			bBusy			=> StartJob, 
			bError			=> Error, 
			nErrId			=> ErrorID);
	
	ELSIF 	SlaveCom[SlaveNo]^.Jobs[JobNo].FunctionCode = 4 THEN
		ReadInputRegs(
			sIPAddr			:= SlaveCom[SlaveNo]^.ipAddr, 
			nTCPPort		:= TO_UINT(SlaveCom[SlaveNo]^.Port), 
			nUnitID			:= SlaveCom[SlaveNo]^.Address, 
			nQuantity		:= SlaveCom[SlaveNo]^.jobs[JobNo].Quantity, 
			nMBAddr			:= SlaveCom[SlaveNo]^.jobs[JobNo].startAddress, 
			cbLength		:= SlaveCom[SlaveNo]^.jobs[JobNo].Quantity * 2, 
			pDestAddr		:= ADR(SlaveCom[SlaveNo]^.Data), 
			bExecute		:= Execute, 
			tTimeout		:= , 
			bBusy			=> StartJob, 
			bError			=> Error, 
			nErrId			=> ErrorID);
	
	ELSIF 	SlaveCom[SlaveNo]^.Jobs[JobNo].FunctionCode = 5 THEN
		WriteSingleCoil(
			sIPAddr			:= SlaveCom[SlaveNo]^.ipAddr, 
			nTCPPort		:= TO_UINT(SlaveCom[SlaveNo]^.Port), 
			nUnitID			:= SlaveCom[SlaveNo]^.Address, 
			nMBAddr			:= SlaveCom[SlaveNo]^.jobs[JobNo].startAddress, 
			nValue			:= SlaveCom[SlaveNo]^.data[1], 
			bExecute		:= Execute, 
			tTimeout		:= , 
			bBusy			=> StartJob, 
			bError			=> Error, 
			nErrId			=> ErrorID);
	
	ELSIF 	SlaveCom[SlaveNo]^.Jobs[JobNo].FunctionCode = 6 THEN
		WriteSingleReg(
			sIPAddr			:= SlaveCom[SlaveNo]^.ipAddr, 
			nTCPPort		:= TO_UINT(SlaveCom[SlaveNo]^.Port), 
			nUnitID			:= SlaveCom[SlaveNo]^.Address, 
			nMBAddr			:= SlaveCom[SlaveNo]^.jobs[JobNo].startAddress, 
			nValue			:= SlaveCom[SlaveNo]^.data[1], 
			bExecute		:= Execute, 
			tTimeout		:= , 
			bBusy			=> StartJob, 
			bError			=> Error, 
			nErrId			=> ErrorID);	
			
	ELSIF 	SlaveCom[SlaveNo]^.Jobs[JobNo].FunctionCode = 8 THEN
		Diagnose(
			sIPAddr			:= SlaveCom[SlaveNo]^.ipAddr, 
			nTCPPort		:= TO_UINT(SlaveCom[SlaveNo]^.Port), 
			nUnitID			:= SlaveCom[SlaveNo]^.Address, 
			bExecute		:= Execute, 
			tTimeout		:= , 
			bBusy			=> StartJob, 
			bError			=> Error, 
			nErrId			=> ErrorID);		

	ELSIF 	SlaveCom[SlaveNo]^.Jobs[JobNo].FunctionCode = 15 THEN
		WriteCoils(
			sIPAddr			:= SlaveCom[SlaveNo]^.ipAddr, 
			nTCPPort		:= TO_UINT(SlaveCom[SlaveNo]^.Port), 
			nUnitID			:= SlaveCom[SlaveNo]^.Address, 
			nQuantity		:= SlaveCom[SlaveNo]^.jobs[JobNo].Quantity, 
			nMBAddr			:= SlaveCom[SlaveNo]^.jobs[JobNo].startAddress, 
			cbLength		:= SlaveCom[SlaveNo]^.jobs[JobNo].Quantity, 
			pSrcAddr		:= ADR(SlaveCom[SlaveNo]^.Data), 
			bExecute		:= Execute, 
			tTimeout		:= , 
			bBusy			=> StartJob, 
			bError			=> Error, 
			nErrId			=> ErrorID);
	
	ELSIF 	SlaveCom[SlaveNo]^.Jobs[JobNo].FunctionCode = 16 THEN
		WriteRegs(
			sIPAddr			:= SlaveCom[SlaveNo]^.ipAddr, 
			nTCPPort		:= TO_UINT(SlaveCom[SlaveNo]^.Port), 
			nUnitID			:= SlaveCom[SlaveNo]^.Address, 
			nQuantity		:= SlaveCom[SlaveNo]^.jobs[JobNo].Quantity, 
			nMBAddr			:= SlaveCom[SlaveNo]^.jobs[JobNo].startAddress, 
			cbLength		:= SlaveCom[SlaveNo]^.jobs[JobNo].Quantity, 
			pSrcAddr		:= ADR(SlaveCom[SlaveNo]^.Data), 
			bExecute		:= Execute, 
			tTimeout		:= , 
			bBusy			=> StartJob, 
			bError			=> Error, 
			nErrId			=> ErrorID);
		
	ELSIF 	SlaveCom[SlaveNo]^.Jobs[JobNo].FunctionCode = 23 THEN
		// not implemented
(*		ReadWriteRegs(
			sIPAddr			:= SlaveCom[SlaveNo]^.ipAddr, 
			nTCPPort		:= SlaveCom[SlaveNo]^.Port, 
			nUnitID			:= SlaveCom[SlaveNo]^.Address, 
			nReadQuantity	:= SlaveCom[SlaveNo]^.jobs[JobNo].Quantity, 
			nMBReadAddr		:= SlaveCom[SlaveNo]^.jobs[JobNo].startAddress, 
			nWriteQuantity	:= , // missing
			nMBWriteAddr	:= , // missing
			cbDestLength	:= SlaveCom[SlaveNo]^.jobs[JobNo].Quantity, 
			pDestAddr		:= ADR(SlaveCom[SlaveNo]^.Data),
			cbSrcLength		:= , // missing
			pSrcAddr 		:= , // missing
			bExecute		:= Execute, 
			tTimeout		:= , 
			bBusy			=> StartJob, 
			bError			=> Error, 
			nErrId			=> ErrorID);	
		*)			
	END_IF
END_METHOD

END_FUNCTION_BLOCK

// ---- POUs/Connectivity/TF625x-Modbus/Master/TF6255-ModbusRtu/ModbusRtuMaster22B.TcPOU
{attribute 'no_check'}
// ModBus comunication master to multible slaves useing RTU protocol
// based on TF6255 - required lib: Tc2_ModbusRTU
FUNCTION_BLOCK ModbusRtuMaster22B
VAR_OUTPUT CONSTANT
	MIN_SLAVE												:	INT := 1;
	MAX_SLAVE												:	INT := PARAM.MODBUS_MAX_SLAVES_OF_MASTER;
{attribute 'displaymode':='binary'}
	OPTION_DISABLE_ERROR_STATE								:	BYTE := 2#0000_0001; //FB will not go into error state and keeps running, even all slaves are in error state
END_VAR
VAR_INPUT
	Enable													:	BOOL ; 		// FB will be processed as long as enable is TRUE 
	ResetTrig												:	BOOL ;		// The function block will be reset with a rising edge 
{attribute 'displaymode':='binary'}
	Options													:	BYTE := 0; //FB options, see VAR_OUTPUT CONSTANT
	SlaveCom												:	ARRAY[MIN_SLAVE..MAX_SLAVE] OF POINTER TO ModbusSlaveCom;
	Timestamp												:	DT;
END_VAR         	
VAR_OUTPUT     
	JobNo													:	INT := 0;
	SlaveNo													:	INT := 0;
{attribute 'displaymode':='binary'}
	SlaveInErrorMask										:	DWORD; //Bit.1 indicates slave 1 in error 	
	Error													:	BOOL;		// Rising edge of Error informs that an error occurred during the execution of the Function Block 
{attribute 'displaymode':='hex'}
	ErrorID													:	MODBUS_ERRORS;		// Error identification - see ADS return codes at Beckhoff infosys for further information 
	ErrorText												:	STRING;
END_VAR
VAR
(* memory **************************************************)
	State 													:	INT := 0;
(* trigger *************************************************)

(* timer ***************************************************)

(* blocks **************************************************)
//	com														:	ModbusRtuMaster_PcCOM := (Timeout := DEFAULT_ADS_TIMEOUT);
	com														:	ModbusRtuMaster_KL6x22B := (Timeout := DEFAULT_ADS_TIMEOUT);
//	com														:	ModbusRtuMaster_KL6x5B := (Timeout := DEFAULT_ADS_TIMEOUT);
(* internal used variables *********************************)
	i,j,k													:	INT :=0;
END_VAR

(* ModBus RTU comunication to multible slaves 	JHue V1.0			*)
(* uncomment necessary master funktion block 						*)
(* use TC2_ModBusRTU.lib											*)
(********************************************************************)

	IF ResetTrig THEN
		reset();
	END_IF
	
	CASE state OF
	0:	(* Idle *)
		IF Enable 
		THEN
			k 												:=	0;
			JobNo  :=  SlaveNo								:=	1;
			state 											:=	10;
		END_IF

	10: 
		IF GetNextSlave() 
		THEN (* find Slave *)
			k 												:= 0;
			IF GetNextJob() 
			THEN (* find JobNo *)
				SlaveCom[SlaveNo]^.currentJobIdx 			:= JobNo;
				SlaveCom[SlaveNo]^.writeJobRequested 		:= SlaveCom[SlaveNo]^.Jobs[JobNo].FunctionCode >= 5;
				State 										:= SEL(SlaveCom[SlaveNo]^.writeJobRequested, 20, 15);
			END_IF
		ELSE
			state 											:=	0;
		END_IF
	
	15: (* wait for valid write date *)
		IF NOT SlaveCom[SlaveNo]^.writeJobRequested
		THEN
			SlaveCom[SlaveNo]^.Jobs[JobNo].Valid 			:= FALSE;
			state 											:= 20;
		END_IF

	20: (* start job *)	
		IF NOT StartJob(FALSE) // Busy
		THEN						
			state 											:= 30;
		END_IF

